VAR_TEMP
  CIP : BOOL ;	//CIP active
  UNIM : BOOL ;	//Unit Not In Maintenance
  GenRel : BOOL ;	//general OK (emergency and maintenance OK)
  EStopOK : BOOL ;	//emergency OK
  UnitNo : INT ;	//unit number
  xTmp : BOOL ;	//Temporary Bool
  iTmp : INT ;	//Temporary INT
  rTmp : REAL ;	//Temporary REAL
  dTmp : DINT ;	//Temporary DINT (free for general use)
  RetValInt : INT ;	//return value
END_VAR
BEGIN
NETWORK
TITLE =General

      SET   ;
// Simulation ---------------------------------------------------------------
      A     DB1511.DBX 1357.7;
      CC    FB  1519; // "U051Sim"
      A     DB1511.DBX   17.3;
      =     DB1511.DBX 1357.7; //Help bit for simulation

// get unit number ----------------------------------------------------------
      L     DB1510.DBW    0;
      T     #UnitNo;

// communication ------------------------------------------------------------
      UC    FB  1515; // U051Com

NETWORK
TITLE =Sequence organisation

      CLR   ;
      =     M    122.2;

// CIP Counter
      CALL FC    29 (
           UnitNo                   := #UnitNo,
           Value                    := DB1515.DBD   54,
           Enable                   := TRUE,
           Down                     := FALSE,
           OriginDetect             := 0.000000e+000,
           MaxDiffPS                := 1.000000e+000,
           SFMRec                   := DB1511.Seq.SFM[15],
           ValueOld                 := DB1511.DBD 1418);

// sequencer ----------------------------------------------------------------
      A     DB1513.DBX   43.1;
      S     DB1513.DBX   97.3;

      CALL FC    40 (
           UnitNo                   := #UnitNo);

END_FUNCTION_BLOCK

FUNCTION_BLOCK FB 1520
TITLE =U052: Water Transfer Plant 12
FAMILY : BOTEC_F1
NAME : UniA
VERSION : 2.1


VAR_TEMP
  EStopOK : BOOL ;	//auxiliary flag
  CIP : BOOL ;	//CIP Program Selected
  xTmp : BOOL ;	//Temporary Bool(free for general use)
  UnitNo : INT ;	//unit number
  UnitFB : INT ;	//unit expansion FB number
  rTmp : REAL ;	//Temporary REAL (free for general use)
  iTmp : INT ;	//Temporary INT (free for general use)
  dTmp : DINT ;	//Temporary DINT (free for general use)
END_VAR
BEGIN
NETWORK
TITLE =general

      CLR   ;
      =     #xTmp;
      =     #EStopOK;

      L     DB1520.DBW    0;
      T     #UnitNo;
      L     DB1520.DBW    2;
      T     #UnitFB;

NETWORK
TITLE =Universal value

      NOP   0;
// unv001 UnV 001 Process Status
      CALL FC    27 (
           UnitNo                   := #UnitNo,
           UnVRec                   := DB2525.unv001,
           ValExt                   := DB2525.DBD  234);

// unv002 UnV 002 Universal Value 02
      CALL FC    27 (
           UnitNo                   := #UnitNo,
           UnVRec                   := DB2525.unv002,
           ValExt                   := DB2525.DBD  362);

// unv003 UnV 003 Universal Value 03
      CALL FC    27 (
           UnitNo                   := #UnitNo,
           UnVRec                   := DB2525.unv003,
           ValExt                   := DB2525.DBD  490);

// unv004 UnV 004 Universal Value 04
      CALL FC    27 (
           UnitNo                   := #UnitNo,
           UnVRec                   := DB2525.unv004,
           ValExt                   := DB2525.DBD  618);

NETWORK
TITLE =special inputs

      NOP   0;
// U52_SpI001 SpI 001 spare
      CALL FC    14 (
           UnitNo                   := #UnitNo,
           SpIRec                   := DB2521.U52_SpI001,
           SpIBit                   := #xTmp);

NETWORK
TITLE =messages

      NOP   0;
// msg001 Msg 001 Message 01
      CALL FC    16 (
           UnitNo                   := #UnitNo,
           MsgRec                   := DB2527.msg001,
           MsgBit                   := DB2527.DBX   82.7);

// msg002 Msg 002 Message 02
      CALL FC    16 (
           UnitNo                   := #UnitNo,
           MsgRec                   := DB2527.msg002,
           MsgBit                   := DB2527.DBX  142.7);

// msg003 Msg 003 Message 03
      CALL FC    16 (
           UnitNo                   := #UnitNo,
           MsgRec                   := DB2527.msg003,
           MsgBit                   := DB2527.DBX  202.7);

NETWORK
TITLE =unit supply

      UC    FB [#UnitFB];

NETWORK
TITLE =Act1  Wasserpumpe
// Act 001
// Box           :
// Input address : #xTmp
// Output address: #xTmp
      CALL FC    70 (
           UnitNo                   := #UnitNo,
           ActRec                   := DB2520.Act1,
           Typ                      := 0,
           FBa                      := I    271.1,
           FBa2                     := #xTmp,
           Out                      := Q    271.1);

NETWORK
TITLE =A12_V11  A12 V11
// Act 002
// Box           : VSA12
// Input address : I260.6
// Output address: Q260.6
      CALL FC    70 (
           UnitNo                   := #UnitNo,
           ActRec                   := DB2520.A12_V11,
           Typ                      := 1,
           FBa                      := #xTmp,
           FBa2                     := I    260.6,
           Out                      := Q    260.6);

NETWORK
TITLE =A12_V12  A12 V12
// Act 003
// Box           : VSA12
// Input address : I260.7
// Output address: Q260.7
      CALL FC    70 (
           UnitNo                   := #UnitNo,
           ActRec                   := DB2520.A12_V12,
           Typ                      := 1,
           FBa                      := #xTmp,
           FBa2                     := I    260.7,
           Out                      := Q    260.7);

NETWORK
TITLE =A12_V13  A12 V13
// Act 004
// Box           : VSA12
// Input address : I261.0
// Output address: Q261.0
      CALL FC    70 (
           UnitNo                   := #UnitNo,
           ActRec                   := DB2520.A12_V13,
           Typ                      := 1,
           FBa                      := #xTmp,
           FBa2                     := I    261.0,
           Out                      := Q    261.0);

NETWORK
TITLE =RV1_A12
// Act 005
// Box           : Ventilinsel 2
// Input address : I321.5
// Output address: Q321.5
      CALL FC    70 (
           UnitNo                   := #UnitNo,
           ActRec                   := DB2520.RV1_A12,
           Typ                      := 1,
           FBa                      := #xTmp,
           FBa2                     := I    321.5,
           Out                      := Q    321.5);

NETWORK
TITLE =RV2_A12
// Act 006
// Box           : Ventilinsel 2
// Input address : I321.6
// Output address: Q321.6
      CALL FC    70 (
           UnitNo                   := #UnitNo,
           ActRec                   := DB2520.RV2_A12,
           Typ                      := 1,
           FBa                      := #xTmp,
           FBa2                     := I    321.6,
           Out                      := Q    321.6);

NETWORK
TITLE =RV3_A12
// Act 007
// Box           : Ventilinsel 2
// Input address : I321.7
// Output address: Q321.7
      CALL FC    70 (
           UnitNo                   := #UnitNo,
           ActRec                   := DB2520.RV3_A12,
           Typ                      := 1,
           FBa                      := #xTmp,
           FBa2                     := I    321.7,
           Out                      := Q    321.7);

NETWORK
TITLE =VR_V4
// Act 008
// Box           : Ventilinsel 4
// Input address : I336.6
// Output address: Q336.6
      CALL FC    70 (
           UnitNo                   := #UnitNo,
           ActRec                   := DB2520.VR_V4,
           Typ                      := 1,
           FBa                      := #xTmp,
           FBa2                     := I    336.6,
           Out                      := Q    336.6);

NETWORK
TITLE =U52_Act010  spare
// Act 010
// Box           :
// Output address: #xtmp
      CALL FC    70 (
           UnitNo                   := #UnitNo,
           ActRec                   := DB2520.U52_Act010,
           Typ                      := 0,
           FBa                      := #xTmp,
           FBa2                     := #xTmp,
           Out                      := #xTmp);

END_FUNCTION_BLOCK

FUNCTION_BLOCK FB 1521
TITLE =U052: Water Transfer Plant 12
FAMILY : BOTEC_F1
NAME : UniE
VERSION : 1.2


VAR_TEMP
  CIP : BOOL ;	//CIP active
  UNIM : BOOL ;	//Unit Not In Maintenance
  GenRel : BOOL ;	//general OK (emergency and maintenance OK)
  EStopOK : BOOL ;	//emergency OK
  UnitNo : INT ;	//unit number
  xTmp : BOOL ;	//Temporary Bool
  iTmp : INT ;	//Temporary INT
  rTmp : REAL ;	//Temporary REAL
  dTmp : DINT ;	//Temporary DINT (free for general use)
  RetValInt : INT ;	//return value
END_VAR
BEGIN
NETWORK
TITLE =General

      SET   ;
// Simulation ---------------------------------------------------------------
      A     DB1521.DBX 1357.7;
      CC    FB  1529; // "U052Sim"
      A     DB1521.DBX   17.3;
      =     DB1521.DBX 1357.7; //Help bit for simulation

// get unit number ----------------------------------------------------------
      L     DB1520.DBW    0;
      T     #UnitNo;

// communication ------------------------------------------------------------
      UC    FB  1525;

NETWORK
TITLE =Sequence organisation

      CLR   ;
      =     M    122.2;

// CIP Counter
      CALL FC    29 (
           UnitNo                   := #UnitNo,
           Value                    := DB1525.DBD   54,
           Enable                   := TRUE,
           Down                     := FALSE,
           OriginDetect             := 0.000000e+000,
           MaxDiffPS                := 1.000000e+000,
           SFMRec                   := DB1521.Seq.SFM[15],
           ValueOld                 := DB1521.DBD 1418);

// sequencer ----------------------------------------------------------------
      A     DB1523.DBX   43.1;
      S     DB1523.DBX   97.3;

      CALL FC    40 (
           UnitNo                   := #UnitNo);

END_FUNCTION_BLOCK

FUNCTION_BLOCK FB 1540
TITLE =U054: Water Transfer Plant 14
FAMILY : BOTEC_F1
NAME : UniA
VERSION : 2.1


VAR_TEMP
  EStopOK : BOOL ;	//auxiliary flag
  CIP : BOOL ;	//CIP Program Selected
  xTmp : BOOL ;	//Temporary Bool(free for general use)
  UnitNo : INT ;	//unit number
  UnitFB : INT ;	//unit expansion FB number
  rTmp : REAL ;	//Temporary REAL (free for general use)
  iTmp : INT ;	//Temporary INT (free for general use)
  dTmp : DINT ;	//Temporary DINT (free for general use)
END_VAR
BEGIN
NETWORK
TITLE =general

      CLR   ;
      =     #xTmp;
      =     #EStopOK;

      L     DB1540.DBW    0;
      T     #UnitNo;
      L     DB1540.DBW    2;
      T     #UnitFB;

NETWORK
TITLE =Universal value

      NOP   0;
// unv001 UnV 001 Process Status
      CALL FC    27 (
           UnitNo                   := #UnitNo,
           UnVRec                   := DB2545.unv001,
           ValExt                   := DB2545.DBD  234);

// unv002 UnV 002 Universal Value 02
      CALL FC    27 (
           UnitNo                   := #UnitNo,
           UnVRec                   := DB2545.unv002,
           ValExt                   := DB2545.DBD  362);

// unv003 UnV 003 Universal Value 03
      CALL FC    27 (
           UnitNo                   := #UnitNo,
           UnVRec                   := DB2545.unv003,
           ValExt                   := DB2545.DBD  490);

// unv004 UnV 004 Universal Value 04
      CALL FC    27 (
           UnitNo                   := #UnitNo,
           UnVRec                   := DB2545.unv004,
           ValExt                   := DB2545.DBD  618);

NETWORK
TITLE =special inputs

      NOP   0;
// U54_SpI001 SpI 001 spare
      CALL FC    14 (
           UnitNo                   := #UnitNo,
           SpIRec                   := DB2541.U54_SpI001,
           SpIBit                   := #xTmp);

NETWORK
TITLE =messages

      NOP   0;
// msg001 Msg 001 Message 01
      CALL FC    16 (
           UnitNo                   := #UnitNo,
           MsgRec                   := DB2547.msg001,
           MsgBit                   := DB2547.DBX   82.7);

// msg002 Msg 002 Message 02
      CALL FC    16 (
           UnitNo                   := #UnitNo,
           MsgRec                   := DB2547.msg002,
           MsgBit                   := DB2547.DBX  142.7);

// msg003 Msg 003 Message 03
      CALL FC    16 (
           UnitNo                   := #UnitNo,
           MsgRec                   := DB2547.msg003,
           MsgBit                   := DB2547.DBX  202.7);

NETWORK
TITLE =unit supply

      UC    FB [#UnitFB];

NETWORK
TITLE =Act1  Wasserpumpe
// Act 001
// Box           :
// Input address : #xTmp
// Output address: #xTmp
      CALL FC    70 (
           UnitNo                   := #UnitNo,
           ActRec                   := DB2540.Act1,
           Typ                      := 0,
           FBa                      := I      6.0,
           FBa2                     := #xTmp,
           Out                      := Q      6.0);

NETWORK
TITLE =A14_V11
// Act 002
// Box           : VSA14
// Input address : I96.6
// Output address: Q96.6
      CALL FC    70 (
           UnitNo                   := #UnitNo,
           ActRec                   := DB2540.A14_V11,
           Typ                      := 1,
           FBa                      := #xTmp,
           FBa2                     := I     96.6,
           Out                      := Q     96.6);

NETWORK
TITLE =A14_V12
// Act 003
// Box           : VSA14
// Input address : I96.7
// Output address: Q96.7
      CALL FC    70 (
           UnitNo                   := #UnitNo,
           ActRec                   := DB2540.A14_V12,
           Typ                      := 1,
           FBa                      := #xTmp,
           FBa2                     := I     96.7,
           Out                      := Q     96.7);

NETWORK
TITLE =A14_V13
// Act 004
// Box           : VSA14
// Input address : I97.0
// Output address: Q97.0
      CALL FC    70 (
           UnitNo                   := #UnitNo,
           ActRec                   := DB2540.A14_V13,
           Typ                      := 1,
           FBa                      := #xTmp,
           FBa2                     := I     97.0,
           Out                      := Q     97.0);

NETWORK
TITLE =RV1_A14
// Act 005
// Box           : Ventilinsel 4
// Input address : I331.5
// Output address: Q331.5
      CALL FC    70 (
           UnitNo                   := #UnitNo,
           ActRec                   := DB2540.RV1_A14,
           Typ                      := 1,
           FBa                      := #xTmp,
           FBa2                     := I    331.5,
           Out                      := Q    331.5);

NETWORK
TITLE =RV2_A14
// Act 006
// Box           : Ventilinsel 4
// Input address : I331.6
// Output address: Q331.6
      CALL FC    70 (
           UnitNo                   := #UnitNo,
           ActRec                   := DB2540.RV2_A14,
           Typ                      := 1,
           FBa                      := #xTmp,
           FBa2                     := I    331.6,
           Out                      := Q    331.6);

NETWORK
TITLE =RV3_A14
// Act 007
// Box           : Ventilinsel 4
// Input address : I331.7
// Output address: Q331.7
      CALL FC    70 (
           UnitNo                   := #UnitNo,
           ActRec                   := DB2540.RV3_A14,
           Typ                      := 1,
           FBa                      := #xTmp,
           FBa2                     := I    331.7,
           Out                      := Q    331.7);

NETWORK
TITLE =VR_V9
// Act 008
// Box           : Ventilinsel 4
// Input address : I336.1
// Output address: Q336.1
      CALL FC    70 (
           UnitNo                   := #UnitNo,
           ActRec                   := DB2540.VR_V9,
           Typ                      := 1,
           FBa                      := #xTmp,
           FBa2                     := I    336.1,
           Out                      := Q    336.1);

NETWORK
TITLE =VR_V8
// Act 009
// Box           : Ventilinsel 4
// Input address : I336.0
// Output address: Q336.0
      CALL FC    70 (
           UnitNo                   := #UnitNo,
           ActRec                   := DB2540.VR_V8,
           Typ                      := 0,//1
           FBa                      := #xTmp,
           FBa2                     := I    336.0,
           Out                      := Q    336.0);

NETWORK
TITLE =A14_V14
// Act 010
// Box           : VSA14
// Input address : I97.1
// Output address: Q97.1
      CALL FC    70 (
           UnitNo                   := #UnitNo,
           ActRec                   := DB2540.A14_V14,
           Typ                      := 0,//1
           FBa                      := #xTmp,
           FBa2                     := I     97.1,
           Out                      := Q     97.1);

END_FUNCTION_BLOCK

FUNCTION_BLOCK FB 1541
TITLE =U054: Water Transfer Plant 14
FAMILY : BOTEC_F1
NAME : UniE
VERSION : 1.2


VAR_TEMP
  CIP : BOOL ;	//CIP active
  UNIM : BOOL ;	//Unit Not In Maintenance
  GenRel : BOOL ;	//general OK (emergency and maintenance OK)
  EStopOK : BOOL ;	//emergency OK
  UnitNo : INT ;	//unit number
  xTmp : BOOL ;	//Temporary Bool
  iTmp : INT ;	//Temporary INT
  rTmp : REAL ;	//Temporary REAL
  dTmp : DINT ;	//Temporary DINT (free for general use)
  RetValInt : INT ;	//return value
END_VAR
BEGIN
NETWORK
TITLE =General

      SET   ;
// Simulation ---------------------------------------------------------------
      A     DB1541.DBX 1357.7;
      CC    FB  1549; // "U054Sim"
      A     DB1541.DBX   17.3;
      =     DB1541.DBX 1357.7; //Help bit for simulation

// get unit number ----------------------------------------------------------
      L     DB1540.DBW    0;
      T     #UnitNo;

// communication ------------------------------------------------------------
      UC    FB  1545; // U054Com

NETWORK
TITLE =Sequence organisation

      CLR   ;
      =     M    122.2;

// CIP Counter
      CALL FC    29 (
           UnitNo                   := #UnitNo,
           Value                    := DB1545.DBD   54,
           Enable                   := TRUE,
           Down                     := FALSE,
           OriginDetect             := 0.000000e+000,
           MaxDiffPS                := 1.000000e+000,
           SFMRec                   := DB1541.Seq.SFM[15],
           ValueOld                 := DB1541.DBD 1418);

// sequencer ----------------------------------------------------------------
      A     DB1543.DBX   43.1;
      S     DB1543.DBX   97.3;

      CALL FC    40 (
           UnitNo                   := #UnitNo);

NETWORK
TITLE =Werte an Mixer



END_FUNCTION_BLOCK

FUNCTION_BLOCK FB 1550
TITLE =U055: Water Transfer Plant 15
FAMILY : BOTEC_F1
NAME : UniA
VERSION : 2.1


VAR_TEMP
  EStopOK : BOOL ;	//auxiliary flag
  CIP : BOOL ;	//CIP Program Selected
  xTmp : BOOL ;	//Temporary Bool(free for general use)
  UnitNo : INT ;	//unit number
  UnitFB : INT ;	//unit expansion FB number
  rTmp : REAL ;	//Temporary REAL (free for general use)
  iTmp : INT ;	//Temporary INT (free for general use)
  dTmp : DINT ;	//Temporary DINT (free for general use)
END_VAR
BEGIN
NETWORK
TITLE =general

      CLR   ;
      =     #xTmp;
      =     #EStopOK;

      L     DB1550.DBW    0;
      T     #UnitNo;
      L     DB1550.DBW    2;
      T     #UnitFB;

NETWORK
TITLE =Universal value

      NOP   0;
// unv001 UnV 001 Process Status
      CALL FC    27 (
           UnitNo                   := #UnitNo,
           UnVRec                   := DB2555.unv001,
           ValExt                   := DB2555.DBD  234);

// unv002 UnV 002 Universal Value 02
      CALL FC    27 (
           UnitNo                   := #UnitNo,
           UnVRec                   := DB2555.unv002,
           ValExt                   := DB2555.DBD  362);

// unv003 UnV 003 Universal Value 03
      CALL FC    27 (
           UnitNo                   := #UnitNo,
           UnVRec                   := DB2555.unv003,
           ValExt                   := DB2555.DBD  490);

// unv004 UnV 004 Universal Value 04
      CALL FC    27 (
           UnitNo                   := #UnitNo,
           UnVRec                   := DB2555.unv004,
           ValExt                   := DB2555.DBD  618);

NETWORK
TITLE =special inputs

      NOP   0;
// U55_SpI001 SpI 001 spare
      CALL FC    14 (
           UnitNo                   := #UnitNo,
           SpIRec                   := DB2551.U55_SpI001,
           SpIBit                   := #xTmp);

NETWORK
TITLE =messages

      NOP   0;
// msg001 Msg 001 Message 01
      CALL FC    16 (
           UnitNo                   := #UnitNo,
           MsgRec                   := DB2557.msg001,
           MsgBit                   := DB2557.DBX   82.7);

// msg002 Msg 002 Message 02
      CALL FC    16 (
           UnitNo                   := #UnitNo,
           MsgRec                   := DB2557.msg002,
           MsgBit                   := DB2557.DBX  142.7);

// msg003 Msg 003 Message 03
      CALL FC    16 (
           UnitNo                   := #UnitNo,
           MsgRec                   := DB2557.msg003,
           MsgBit                   := DB2557.DBX  202.7);

NETWORK
TITLE =unit supply

      UC    FB [#UnitFB];

NETWORK
TITLE =Act1  Wasserpumpe
// Act 001
// Box           :
// Input address : #xTmp
// Output address: #xTmp
      CALL FC    70 (
           UnitNo                   := #UnitNo,
           ActRec                   := DB2550.Act1,
           Typ                      := 3,
           FBa                      := #xTmp,
           FBa2                     := #xTmp,
           Out                      := #xTmp);

NETWORK
TITLE =RV1_A15
// Act 005
// Box           : Ventilinsel 4
// Input address : I333.5
// Output address: Q333.5
      CALL FC    70 (
           UnitNo                   := #UnitNo,
           ActRec                   := DB2550.RV1_A15,
           Typ                      := 1,
           FBa                      := #xTmp,
           FBa2                     := I    333.5,
           Out                      := Q    333.5);

NETWORK
TITLE =RV2_A15
// Act 006
// Box           : Ventilinsel 4
// Input address : I333.6
// Output address: Q333.6
      CALL FC    70 (
           UnitNo                   := #UnitNo,
           ActRec                   := DB2550.RV2_A15,
           Typ                      := 1,
           FBa                      := #xTmp,
           FBa2                     := I    333.6,
           Out                      := Q    333.6);

NETWORK
TITLE =RV3_A15
// Act 007
// Box           : Ventilinsel 4
// Input address : I333.7
// Output address: Q333.7
      CALL FC    70 (
           UnitNo                   := #UnitNo,
           ActRec                   := DB2550.RV3_A15,
           Typ                      := 1,
           FBa                      := #xTmp,
           FBa2                     := I    333.7,
           Out                      := Q    333.7);

NETWORK
TITLE =U55_Act010  spare
// Act 010
// Box           :
// Output address: #xtmp
      CALL FC    70 (
           UnitNo                   := #UnitNo,
           ActRec                   := DB2550.U55_Act010,
           Typ                      := 0,
           FBa                      := #xTmp,
           FBa2                     := #xTmp,
           Out                      := #xTmp);

END_FUNCTION_BLOCK

FUNCTION_BLOCK FB 1551
TITLE =U055: Water Transfer Plant 15
FAMILY : BOTEC_F1
NAME : UniE
VERSION : 1.2


VAR_TEMP
  CIP : BOOL ;	//CIP active
  UNIM : BOOL ;	//Unit Not In Maintenance
  GenRel : BOOL ;	//general OK (emergency and maintenance OK)
  EStopOK : BOOL ;	//emergency OK
  UnitNo : INT ;	//unit number
  xTmp : BOOL ;	//Temporary Bool
  iTmp : INT ;	//Temporary INT
  rTmp : REAL ;	//Temporary REAL
  dTmp : DINT ;	//Temporary DINT (free for general use)
  RetValInt : INT ;	//return value
END_VAR
BEGIN
NETWORK
TITLE =General

      SET   ;
// Simulation ---------------------------------------------------------------
      A     DB1551.DBX 1357.7;
      CC    FB  1559; // "U055Sim"
      A     DB1551.DBX   17.3;
      =     DB1551.DBX 1357.7; //Help bit for simulation

// get unit number ----------------------------------------------------------
      L     DB1550.DBW    0;
      T     #UnitNo;

// communication ------------------------------------------------------------
      UC    FB  1555; // U055Com

NETWORK
TITLE =Sequence organisation

      CLR   ;
      =     M    122.2;

// CIP Counter
      CALL FC    29 (
           UnitNo                   := #UnitNo,
           Value                    := DB1555.DBD   54,
           Enable                   := TRUE,
           Down                     := FALSE,
           OriginDetect             := 0.000000e+000,
           MaxDiffPS                := 1.000000e+000,
           SFMRec                   := DB1551.Seq.SFM[15],
           ValueOld                 := DB1551.DBD 1418);

// sequencer ----------------------------------------------------------------
      A     DB1553.DBX   43.1;
      S     DB1553.DBX   97.3;

      CALL FC    40 (
           UnitNo                   := #UnitNo);

END_FUNCTION_BLOCK

FUNCTION_BLOCK FB 1560
TITLE =U056: Fresh Water Transfer
FAMILY : BOTEC_F1
NAME : UniA
VERSION : 2.1


VAR_TEMP
  EStopOK : BOOL ;	//auxiliary flag
  CIP : BOOL ;	//CIP Program Selected
  xTmp : BOOL ;	//Temporary Bool(free for general use)
  UnitNo : INT ;	//unit number
  UnitFB : INT ;	//unit expansion FB number
  rTmp : REAL ;	//Temporary REAL (free for general use)
  iTmp : INT ;	//Temporary INT (free for general use)
  dTmp : DINT ;	//Temporary DINT (free for general use)
END_VAR
BEGIN
NETWORK
TITLE =general

      CLR   ;
      =     #xTmp;
      =     #EStopOK;

      L     DB1560.DBW    0;
      T     #UnitNo;
      L     DB1560.DBW    2;
      T     #UnitFB;

NETWORK
TITLE =Universal value

      NOP   0;
// unv001 UnV 001 Process Status
      CALL FC    27 (
           UnitNo                   := #UnitNo,
           UnVRec                   := DB2565.unv001,
           ValExt                   := DB2565.DBD  234);

// unv002 UnV 002 Universal Value 02
      CALL FC    27 (
           UnitNo                   := #UnitNo,
           UnVRec                   := DB2565.unv002,
           ValExt                   := DB2565.DBD  362);

// unv003 UnV 003 Universal Value 03
      CALL FC    27 (
           UnitNo                   := #UnitNo,
           UnVRec                   := DB2565.unv003,
           ValExt                   := DB2565.DBD  490);

// unv004 UnV 004 Universal Value 04
      CALL FC    27 (
           UnitNo                   := #UnitNo,
           UnVRec                   := DB2565.unv004,
           ValExt                   := DB2565.DBD  618);

NETWORK
TITLE =messages

      NOP   0;
// msg001 Msg 001 Message 01
      CALL FC    16 (
           UnitNo                   := #UnitNo,
           MsgRec                   := DB2567.msg001,
           MsgBit                   := DB2567.DBX   82.7);

// msg002 Msg 002 Message 02
      CALL FC    16 (
           UnitNo                   := #UnitNo,
           MsgRec                   := DB2567.msg002,
           MsgBit                   := DB2567.DBX  142.7);

// msg003 Msg 003 Message 03
      CALL FC    16 (
           UnitNo                   := #UnitNo,
           MsgRec                   := DB2567.msg003,
           MsgBit                   := DB2567.DBX  202.7);

NETWORK
TITLE =unit supply

      UC    FB [#UnitFB];

NETWORK
TITLE =FW_P1  FWP1 Pumpe Frischwasser
// Act 001
// Box           : S6 U6.3
// Input address : I6.7
// Output address: Q6.7
      CALL FC    70 (
           UnitNo                   := #UnitNo,
           ActRec                   := DB2560.FW_P1,
           Typ                      := 1,
           FBa                      := #xTmp,
           FBa2                     := I      6.7,
           Out                      := Q      6.7);

NETWORK
TITLE =FW_RV2
// Act 006
// Box           : Ventilinsel 5
// Input address : I339.5
// Output address: Q339.5
      CALL FC    70 (
           UnitNo                   := #UnitNo,
           ActRec                   := DB2560.FW_RV2,
           Typ                      := 1,
           FBa                      := #xTmp,
           FBa2                     := I    339.5,
           Out                      := Q    339.5);

END_FUNCTION_BLOCK

FUNCTION_BLOCK FB 1561
TITLE =U056: Fresh Water Transfer
FAMILY : BOTEC_F1
NAME : UniE
VERSION : 1.2


VAR_TEMP
  CIP : BOOL ;	//CIP active
  UNIM : BOOL ;	//Unit Not In Maintenance
  GenRel : BOOL ;	//general OK (emergency and maintenance OK)
  EStopOK : BOOL ;	//emergency OK
  UnitNo : INT ;	//unit number
  xTmp : BOOL ;	//Temporary Bool
  iTmp : INT ;	//Temporary INT
  rTmp : REAL ;	//Temporary REAL
  dTmp : DINT ;	//Temporary DINT (free for general use)
  RetValInt : INT ;	//return value
END_VAR
BEGIN
NETWORK
TITLE =General

      SET   ;
// Simulation ---------------------------------------------------------------
      A     DB1561.DBX 1357.7;
      CC    FB  1569; // "U056Sim"
      A     DB1561.DBX   17.3;
      =     DB1561.DBX 1357.7; //Help bit for simulation

// get unit number ----------------------------------------------------------
      L     DB1560.DBW    0;
      T     #UnitNo;

// CIP ----------------------------------------------------------------------
      L     DB1561.DBD   54;
      L     0;
      <D    ;
      =     #CIP;

// emergency OK -------------------------------------------------------------
      A     DB1565.DBX   27.0; //Emergency Stop OK
      =     #EStopOK;

// Write Unit in Maintenance ------------------------------------------------

      AN    DB1561.DBX   69.7;
      =     #UNIM;

// emergency and maintenance OK ---------------------------------------------
      A     #EStopOK;
      A     #UNIM;
      =     #GenRel;

// communication ------------------------------------------------------------
      UC    FB  1565; // U056Com

NETWORK
TITLE =Universal Value

      NOP   0;

// ----------------------------------------------------------
// unv001 Process Status
// ----------------------------------------------------------
// process value to UnV
//      L     0.000000e+000
//      T     "U056UnVD".unv001.ValExt

// ----------------------------------------------------------
// unv002 Universal Value 02
// ----------------------------------------------------------
// process value to UnV
//      L     0.000000e+000
//      T     "U056UnVD".unv002.ValExt

// ----------------------------------------------------------
// unv003 Universal Value 03
// ----------------------------------------------------------
// process value to UnV
//      L     0.000000e+000
//      T     "U056UnVD".unv003.ValExt

// ----------------------------------------------------------
// unv004 Universal Value 04
// ----------------------------------------------------------
// process value to UnV
//      L     0.000000e+000
//      T     "U056UnVD".unv004.ValExt

NETWORK
TITLE =Messages

      NOP   0;

// ----------------------------------------------------------
// msg001 Message 01
// ----------------------------------------------------------
      SET   ;
      R     DB2567.DBX   80.7;
      =     DB2567.DBX   81.4;

      CLR   ;
      =     DB2567.DBX   82.7;

// ----------------------------------------------------------
// msg002 Message 02
// ----------------------------------------------------------
      SET   ;
      R     DB2567.DBX  140.7;
      =     DB2567.DBX  141.4;

      CLR   ;
      =     DB2567.DBX  142.7;

// ----------------------------------------------------------
// msg003 Message 03
// ----------------------------------------------------------
      SET   ;
      R     DB2567.DBX  200.7;
      =     DB2567.DBX  201.4;

      CLR   ;
      =     DB2567.DBX  202.7;

NETWORK
TITLE =Sequence organisation

      CLR   ;
      =     M    122.2;

// SFM supply ----------------------------------------------------------------

// sequencer ----------------------------------------------------------------
      A     DB1563.DBX   43.1;
      S     DB1563.DBX   97.3;

      CALL FC    40 (
           UnitNo                   := #UnitNo);

NETWORK
TITLE =Auto / Manual

      SET   ;
      AN    M    122.2;
      JC    MODE;
      AN    M    120.1;

// assign actuator mode
      AN    M    120.1;
      =     DB2560.DBX  105.4;
      =     DB2560.DBX  505.4;


MODE: SET   ;

NETWORK
TITLE =FW_P1 FWP1 Pumpe Frischwasser

      A     #GenRel;
      A     DB2560.DBX  106.7;
      =     DB2560.DBX  107.6;
END_FUNCTION_BLOCK

FUNCTION_BLOCK FB 1570
TITLE =U057: Water Transfer Brewhouse
FAMILY : BOTEC_F1
NAME : UniA
VERSION : 2.1


VAR_TEMP
  EStopOK : BOOL ;	//auxiliary flag
  CIP : BOOL ;	//CIP Program Selected
  xTmp : BOOL ;	//Temporary Bool(free for general use)
  UnitNo : INT ;	//unit number
  UnitFB : INT ;	//unit expansion FB number
  rTmp : REAL ;	//Temporary REAL (free for general use)
  iTmp : INT ;	//Temporary INT (free for general use)
  dTmp : DINT ;	//Temporary DINT (free for general use)
END_VAR
BEGIN
NETWORK
TITLE =general

      CLR   ;
      =     #xTmp;
      =     #EStopOK;

      L     DB1570.DBW    0;
      T     #UnitNo;
      L     DB1570.DBW    2;
      T     #UnitFB;

NETWORK
TITLE =Universal value

      NOP   0;
// unv001 UnV 001 Process Status
      CALL FC    27 (
           UnitNo                   := #UnitNo,
           UnVRec                   := DB2575.unv001,
           ValExt                   := DB2575.DBD  234);

// unv002 UnV 002 Universal Value 02
      CALL FC    27 (
           UnitNo                   := #UnitNo,
           UnVRec                   := DB2575.unv002,
           ValExt                   := DB2575.DBD  362);

// unv003 UnV 003 Universal Value 03
      CALL FC    27 (
           UnitNo                   := #UnitNo,
           UnVRec                   := DB2575.unv003,
           ValExt                   := DB2575.DBD  490);

// unv004 UnV 004 Universal Value 04
      CALL FC    27 (
           UnitNo                   := #UnitNo,
           UnVRec                   := DB2575.unv004,
           ValExt                   := DB2575.DBD  618);

NETWORK
TITLE =special inputs

      NOP   0;
// AB_SH_DT_LAMPEN_PRUEFEN SpI 002 AUSSENBEDIENUNG SUDHAUS
      CALL FC    14 (
           UnitNo                   := #UnitNo,
           SpIRec                   := DB2571.AB_SH_DT_LAMPEN_PRUEFEN,
           SpIBit                   := I     14.5);

// AB_SH_LDT_WASSER_OPUMP SpI 003 AUSSENBEDIENUNG SUDHAUS
      CALL FC    14 (
           UnitNo                   := #UnitNo,
           SpIRec                   := DB2571.AB_SH_LDT_WASSER_OPUMP,
           SpIBit                   := I     14.6);

// AB_SH_LDT_WASSER_MPUMP SpI 004 AUSSEN SUDHAUS
      CALL FC    14 (
           UnitNo                   := #UnitNo,
           SpIRec                   := DB2571.AB_SH_LDT_WASSER_MPUMP,
           SpIBit                   := I     15.3);

// AB_SH_DT_START SpI 005 AUSSENBEDIENUNG SUDHAUS
      CALL FC    14 (
           UnitNo                   := #UnitNo,
           SpIRec                   := DB2571.AB_SH_DT_START,
           SpIBit                   := I     15.6);

// AB_SH_DT_STOP SpI 006 AUSSENBEDIENUNG SUDHAUS
      CALL FC    14 (
           UnitNo                   := #UnitNo,
           SpIRec                   := DB2571.AB_SH_DT_STOP,
           SpIBit                   := I     15.7);

NETWORK
TITLE =messages

      NOP   0;
// msg001 Msg 001 Message 01
      CALL FC    16 (
           UnitNo                   := #UnitNo,
           MsgRec                   := DB2577.msg001,
           MsgBit                   := DB2577.DBX   82.7);

// msg002 Msg 002 Message 02
      CALL FC    16 (
           UnitNo                   := #UnitNo,
           MsgRec                   := DB2577.msg002,
           MsgBit                   := DB2577.DBX  142.7);

// msg003 Msg 003 Message 03
      CALL FC    16 (
           UnitNo                   := #UnitNo,
           MsgRec                   := DB2577.msg003,
           MsgBit                   := DB2577.DBX  202.7);

NETWORK
TITLE =unit supply

      UC    FB [#UnitFB];

NETWORK
TITLE =SH_P1  SHP1
// Act 001
// Box           : S6 U6.3
// Input address : I6.4
// Output address: Q6.4
      CALL FC    70 (
           UnitNo                   := #UnitNo,
           ActRec                   := DB2570.SH_P1,
           Typ                      := 1,
           FBa                      := #xTmp,
           FBa2                     := I      6.4,
           Out                      := Q      6.4);

NETWORK
TITLE =AB_SH_LAMPE_LDT_WASSOP  Lampe AUSSEN SUDHAUS (ohne Pumpe)
// Act 002
// Box           : S6 U6.3
// Output address: Q14.6
      CALL FC    70 (
           UnitNo                   := #UnitNo,
           ActRec                   := DB2570.AB_SH_LAMPE_LDT_WASSOP,
           Typ                      := 0,
           FBa                      := #xTmp,
           FBa2                     := #xTmp,
           Out                      := Q     14.6);

NETWORK
TITLE =AB_SH_LAMPE_FREIGWASSER  Lampe AUSSENBEDIENUNG SUDHAUS (Freigabe
// Act 003
// Box           : S6 U6.3
// Output address: Q14.7
      CALL FC    70 (
           UnitNo                   := #UnitNo,
           ActRec                   := DB2570.AB_SH_LAMPE_FREIGWASSER,
           Typ                      := 0,
           FBa                      := #xTmp,
           FBa2                     := #xTmp,
           Out                      := Q     14.7);

NETWORK
TITLE =AB_SH_LAMPE_LDT_WASSMP  Lampe AUSSENBEDIENUNG SUDHAUS (mit Pumpe
// Act 004
// Box           : S6 U6.3
// Output address: Q15.0
      CALL FC    70 (
           UnitNo                   := #UnitNo,
           ActRec                   := DB2570.AB_SH_LAMPE_LDT_WASSMP,
           Typ                      := 0,
           FBa                      := #xTmp,
           FBa2                     := #xTmp,
           Out                      := Q     15.0);

NETWORK
TITLE =BH_RV2
// Act 006
// Box           : Ventilinsel 5
// Input address : I339.6
// Output address: Q339.6
      CALL FC    70 (
           UnitNo                   := #UnitNo,
           ActRec                   := DB2570.BH_RV2,
           Typ                      := 1,
           FBa                      := #xTmp,
           FBa2                     := I    339.6,
           Out                      := Q    339.6);

END_FUNCTION_BLOCK

FUNCTION_BLOCK FB 1571
TITLE =U057: Water Transfer Brewhouse
FAMILY : BOTEC_F1
NAME : UniE
VERSION : 1.2


VAR_TEMP
  CIP : BOOL ;	//CIP active
  UNIM : BOOL ;	//Unit Not In Maintenance
  GenRel : BOOL ;	//general OK (emergency and maintenance OK)
  EStopOK : BOOL ;	//emergency OK
  UnitNo : INT ;	//unit number
  xTmp : BOOL ;	//Temporary Bool
  iTmp : INT ;	//Temporary INT
  rTmp : REAL ;	//Temporary REAL
  dTmp : DINT ;	//Temporary DINT (free for general use)
  RetValInt : INT ;	//return value
END_VAR
BEGIN
NETWORK
TITLE =General

      SET   ;
// Simulation ---------------------------------------------------------------
      A     DB1571.DBX 1357.7;
      CC    FB  1579; // "U057Sim"
      A     DB1571.DBX   17.3;
      =     DB1571.DBX 1357.7; //Help bit for simulation

// get unit number ----------------------------------------------------------
      L     DB1570.DBW    0;
      T     #UnitNo;

// CIP ----------------------------------------------------------------------
      L     DB1571.DBD   54;
      L     0;
      <D    ;
      =     #CIP;

// emergency OK -------------------------------------------------------------
      A     DB1575.DBX   27.0; //Emergency Stop OK
      =     #EStopOK;

// Write Unit in Maintenance ------------------------------------------------

      AN    DB1571.DBX   69.7;
      =     #UNIM;

// emergency and maintenance OK ---------------------------------------------
      A     #EStopOK;
      A     #UNIM;
      =     #GenRel;

// communication ------------------------------------------------------------
      UC    FB  1575; // U057Com

NETWORK
TITLE =Universal Value

      NOP   0;

// ----------------------------------------------------------
// unv001 Process Status
// ----------------------------------------------------------
// process value to UnV
//      L     0.000000e+000
//      T     "U057UnVD".unv001.ValExt

// ----------------------------------------------------------
// unv002 Universal Value 02
// ----------------------------------------------------------
// process value to UnV
//      L     0.000000e+000
//      T     "U057UnVD".unv002.ValExt

// ----------------------------------------------------------
// unv003 Universal Value 03
// ----------------------------------------------------------
// process value to UnV
//      L     0.000000e+000
//      T     "U057UnVD".unv003.ValExt

// ----------------------------------------------------------
// unv004 Universal Value 04
// ----------------------------------------------------------
// process value to UnV
//      L     0.000000e+000
//      T     "U057UnVD".unv004.ValExt

NETWORK
TITLE =Special Input

      NOP   0;

// ----------------------------------------------------------
// AB_SH_DT_LAMPEN_PRUEFEN AUSSENBEDIENUNG SUDHAUS
// ----------------------------------------------------------
      CLR   ;
//      =     "U057SpID".AB_SH_DT_LAMPEN_PRUEFEN.EAl
//      =     "U057SpID".AB_SH_DT_LAMPEN_PRUEFEN.Pre

// ----------------------------------------------------------
// AB_SH_LDT_WASSER_OPUMP AUSSENBEDIENUNG SUDHAUS
// ----------------------------------------------------------
      CLR   ;
//      =     "U057SpID".AB_SH_LDT_WASSER_OPUMP.EAl
//      =     "U057SpID".AB_SH_LDT_WASSER_OPUMP.Pre

// ----------------------------------------------------------
// AB_SH_LDT_WASSER_MPUMP AUSSENBEDIENUNG SUDHAUS
// ----------------------------------------------------------
      CLR   ;
//      =     "U057SpID".AB_SH_LDT_WASSER_MPUMP.EAl
//      =     "U057SpID".AB_SH_LDT_WASSER_MPUMP.Pre

// ----------------------------------------------------------
// AB_SH_DT_START AUSSENBEDIENUNG SUDHAUS
// ----------------------------------------------------------
      CLR   ;
//      =     "U057SpID".AB_SH_DT_START.EAl
//      =     "U057SpID".AB_SH_DT_START.Pre

// ----------------------------------------------------------
// AB_SH_DT_STOP AUSSENBEDIENUNG SUDHAUS
// ----------------------------------------------------------
      CLR   ;
//      =     "U057SpID".AB_SH_DT_STOP.EAl
//      =     "U057SpID".AB_SH_DT_STOP.Pre

NETWORK
TITLE =Messages

      NOP   0;

// ----------------------------------------------------------
// msg001 Message 01
// ----------------------------------------------------------
      SET   ;
      R     DB2577.DBX   80.7;
      =     DB2577.DBX   81.4;

      CLR   ;
      =     DB2577.DBX   82.7;

// ----------------------------------------------------------
// msg002 Message 02
// ----------------------------------------------------------
      SET   ;
      R     DB2577.DBX  140.7;
      =     DB2577.DBX  141.4;

      CLR   ;
      =     DB2577.DBX  142.7;

// ----------------------------------------------------------
// msg003 Message 03
// ----------------------------------------------------------
      SET   ;
      R     DB2577.DBX  200.7;
      =     DB2577.DBX  201.4;

      CLR   ;
      =     DB2577.DBX  202.7;

NETWORK
TITLE =Sequence organisation


// SFM supply ----------------------------------------------------------------

// sequencer ----------------------------------------------------------------
      A     DB1573.DBX   43.1;
      S     DB1573.DBX   97.3;

      CALL FC    40 (
           UnitNo                   := #UnitNo);

NETWORK
TITLE =Auto / Manual

      SET   ;
      AN    M    122.2;
      JC    MODE;
      AN    M    120.1;

// assign actuator mode
      AN    M    120.1;
      =     DB2570.DBX  105.4;
      =     DB2570.DBX  185.4;
      =     DB2570.DBX  265.4;
      =     DB2570.DBX  345.4;

      =     DB2570.DBX  425.4;
      =     DB2570.DBX  505.4;




MODE: SET   ;

NETWORK
TITLE =SH_P1 SHP1
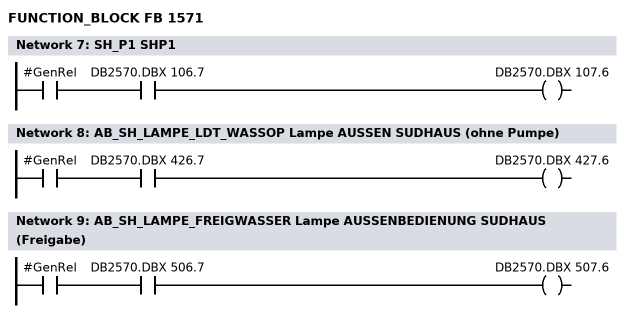

      A     #GenRel;
      A     DB2570.DBX  106.7;
      =     DB2570.DBX  107.6;
NETWORK
TITLE =AB_SH_LAMPE_LDT_WASSOP Lampe AUSSEN SUDHAUS (ohne Pumpe)

      A     #GenRel;
      A     DB2570.DBX  426.7;
      =     DB2570.DBX  427.6;
NETWORK
TITLE =AB_SH_LAMPE_FREIGWASSER Lampe AUSSENBEDIENUNG SUDHAUS (Freigabe)

      A     #GenRel;
      A     DB2570.DBX  506.7;
      =     DB2570.DBX  507.6;
END_FUNCTION_BLOCK

FUNCTION_BLOCK FB 1580
TITLE =U058: Water Transfer Syrup
FAMILY : BOTEC_F1
NAME : UniA
VERSION : 2.1


VAR_TEMP
  EStopOK : BOOL ;	//auxiliary flag
  CIP : BOOL ;	//CIP Program Selected
  xTmp : BOOL ;	//Temporary Bool(free for general use)
  UnitNo : INT ;	//unit number
  UnitFB : INT ;	//unit expansion FB number
  rTmp : REAL ;	//Temporary REAL (free for general use)
  iTmp : INT ;	//Temporary INT (free for general use)
  dTmp : DINT ;	//Temporary DINT (free for general use)
END_VAR
BEGIN
NETWORK
TITLE =general

      CLR   ;
      =     #xTmp;
      =     #EStopOK;

      L     DB1580.DBW    0;
      T     #UnitNo;
      L     DB1580.DBW    2;
      T     #UnitFB;

NETWORK
TITLE =analog inputs

      NOP   0;
// SRW_PIC1 AnI 001
      CALL FC    24 (
           UnitNo                   := #UnitNo,
           AnIRec                   := DB2583.SRW_PIC1,
           ValPer                   := IW   516);

NETWORK
TITLE =Universal value

      NOP   0;
// unv001 UnV 001 Process Status
      CALL FC    27 (
           UnitNo                   := #UnitNo,
           UnVRec                   := DB2585.unv001,
           ValExt                   := DB2585.DBD  234);

// unv002 UnV 002 Universal Value 02
      CALL FC    27 (
           UnitNo                   := #UnitNo,
           UnVRec                   := DB2585.unv002,
           ValExt                   := DB2585.DBD  362);

// unv003 UnV 003 Universal Value 03
      CALL FC    27 (
           UnitNo                   := #UnitNo,
           UnVRec                   := DB2585.unv003,
           ValExt                   := DB2585.DBD  490);

// unv004 UnV 004 Universal Value 04
      CALL FC    27 (
           UnitNo                   := #UnitNo,
           UnVRec                   := DB2585.unv004,
           ValExt                   := DB2585.DBD  618);

NETWORK
TITLE =special inputs

      NOP   0;
// SW_FS1 SpI 002 Flussschalter Wasserpumpe Sirupraum
      CALL FC    14 (
           UnitNo                   := #UnitNo,
           SpIRec                   := DB2581.SW_FS1,
           SpIBit                   := I    188.0);

// WAS_Anforderung SpI 003 Anforderung Wasser
      CALL FC    14 (
           UnitNo                   := #UnitNo,
           SpIRec                   := DB2581.WAS_Anforderung,
           SpIBit                   := DB1585.DBX   26.3);

NETWORK
TITLE =messages

      NOP   0;
// msg001 Msg 001 Message 01
      CALL FC    16 (
           UnitNo                   := #UnitNo,
           MsgRec                   := DB2587.msg001,
           MsgBit                   := DB2587.DBX   82.7);

// msg002 Msg 002 Message 02
      CALL FC    16 (
           UnitNo                   := #UnitNo,
           MsgRec                   := DB2587.msg002,
           MsgBit                   := DB2587.DBX  142.7);

// msg003 Msg 003 Message 03
      CALL FC    16 (
           UnitNo                   := #UnitNo,
           MsgRec                   := DB2587.msg003,
           MsgBit                   := DB2587.DBX  202.7);

NETWORK
TITLE =controllers

      NOP   0;
// SR_P1_PID PID 001 Druckregelung Sirupwasser SR.P1
      CALL FC    55 (
           UnitNo                   := #UnitNo,
           PIDRec                   := DB2586.SR_P1_PID,
           SpExt                    := DB2586.DBD  234,
           PVal                     := DB2586.DBD  254,
           OPer                     := PQW  516);

NETWORK
TITLE =unit supply

      UC    FB [#UnitFB];

NETWORK
TITLE =SR_P1  Wasserpumpe Sirupraum
// Act 001
// Box           : VSSK
// Input address : I73.7
// Output address: Q53.7
      CALL FC    70 (
           UnitNo                   := #UnitNo,
           ActRec                   := DB2580.SR_P1,
           Typ                      := 3,
           FBa                      := I     73.7,
           FBa2                     := #xTmp,
           Out                      := Q     53.7);

NETWORK
TITLE =WAS_Bereit  Wasser kann agefordert werden
// Act 002
// Box           : Sirup
// Output address: DB_SEND_DOEHLER.Wasser.Bereit
      CALL FC    70 (
           UnitNo                   := #UnitNo,
           ActRec                   := DB2580.WAS_Bereit,
           Typ                      := 0,
           FBa                      := #xTmp,
           FBa2                     := #xTmp,
           Out                      := DB404.DBX    2.0);

NETWORK
TITLE =WAS_Pumpe_laeuft  Die Wasserpumpe laeuft
// Act 003
// Box           : Sirup
// Output address: DB_SEND_DOEHLER.Wasser.Pumpe_laeuft
      CALL FC    70 (
           UnitNo                   := #UnitNo,
           ActRec                   := DB2580.WAS_Pumpe_laeuft,
           Typ                      := 0,
           FBa                      := #xTmp,
           FBa2                     := #xTmp,
           Out                      := DB404.DBX    2.1);

NETWORK
TITLE =SK_RV2
// Act 006
// Box           : Ventilinsel 5
// Input address : I339.4
// Output address: Q339.4
      CALL FC    70 (
           UnitNo                   := #UnitNo,
           ActRec                   := DB2580.SK_RV2,
           Typ                      := 1,
           FBa                      := #xTmp,
           FBa2                     := I    339.4,
           Out                      := Q    339.4);

END_FUNCTION_BLOCK

FUNCTION_BLOCK FB 1581
TITLE =U058: Water Transfer Syrup
FAMILY : BOTEC_F1
NAME : UniE
VERSION : 1.2


VAR_TEMP
  CIP : BOOL ;	//CIP active
  UNIM : BOOL ;	//Unit Not In Maintenance
  GenRel : BOOL ;	//general OK (emergency and maintenance OK)
  EStopOK : BOOL ;	//emergency OK
  UnitNo : INT ;	//unit number
  xTmp : BOOL ;	//Temporary Bool
  iTmp : INT ;	//Temporary INT
  rTmp : REAL ;	//Temporary REAL
  dTmp : DINT ;	//Temporary DINT (free for general use)
  RetValInt : INT ;	//return value
END_VAR
BEGIN
NETWORK
TITLE =General

      SET   ;
// Simulation ---------------------------------------------------------------
      A     DB1581.DBX 1357.7;
      CC    FB  1589; // "U058Sim"
      A     DB1581.DBX   17.3;
      =     DB1581.DBX 1357.7; //Help bit for simulation

// get unit number ----------------------------------------------------------
      L     DB1580.DBW    0;
      T     #UnitNo;

// CIP ----------------------------------------------------------------------
      L     DB1581.DBD   54;
      L     0;
      <D    ;
      =     #CIP;

// emergency OK -------------------------------------------------------------
      A     DB1585.DBX   27.0; //Emergency Stop OK
      =     #EStopOK;

// Write Unit in Maintenance ------------------------------------------------

      AN    DB1581.DBX   69.7;
      =     #UNIM;

// emergency and maintenance OK ---------------------------------------------
      A     #EStopOK;
      A     #UNIM;
      =     #GenRel;

// communication ------------------------------------------------------------
      UC    FB  1585; // U058Com

NETWORK
TITLE =Analog Inputs

      NOP   0;

// ----------------------------------------------------------
// SRW_PIC1
// ----------------------------------------------------------
      L     DB1581.DBD 1118; // !!! insert correct SFM !!!
      T     DB2583.DBD  238;

      SET   ;
      =     DB2583.DBX  141.5;

NETWORK
TITLE =Universal Value

      NOP   0;

// ----------------------------------------------------------
// unv001 Process Status
// ----------------------------------------------------------
// process value to UnV
//      L     0.000000e+000
//      T     "U058UnVD".unv001.ValExt

// ----------------------------------------------------------
// unv002 Universal Value 02
// ----------------------------------------------------------
// process value to UnV
//      L     0.000000e+000
//      T     "U058UnVD".unv002.ValExt

// ----------------------------------------------------------
// unv003 Universal Value 03
// ----------------------------------------------------------
// process value to UnV
//      L     0.000000e+000
//      T     "U058UnVD".unv003.ValExt

// ----------------------------------------------------------
// unv004 Universal Value 04
// ----------------------------------------------------------
// process value to UnV
//      L     0.000000e+000
//      T     "U058UnVD".unv004.ValExt

NETWORK
TITLE =Special Input

      NOP   0;

// ----------------------------------------------------------
// SW_FS1 Flussschalter Wasserpumpe Sirupraum
// ----------------------------------------------------------
      A     DB2580.DBX  102.6;
      =     DB2581.DBX  141.4;
      =     DB2581.DBX  141.5;

// ----------------------------------------------------------
// WAS_Anforderung Anforderung Wasser
// ----------------------------------------------------------
      CLR   ;
      =     DB2581.DBX  201.4;
      =     DB2581.DBX  201.5;

NETWORK
TITLE =Messages

      NOP   0;

// ----------------------------------------------------------
// msg001 Message 01
// ----------------------------------------------------------
      SET   ;
      R     DB2587.DBX   80.7;
      =     DB2587.DBX   81.4;

      CLR   ;
      =     DB2587.DBX   82.7;

// ----------------------------------------------------------
// msg002 Message 02
// ----------------------------------------------------------
      SET   ;
      R     DB2587.DBX  140.7;
      =     DB2587.DBX  141.4;

      CLR   ;
      =     DB2587.DBX  142.7;

// ----------------------------------------------------------
// msg003 Message 03
// ----------------------------------------------------------
      SET   ;
      R     DB2587.DBX  200.7;
      =     DB2587.DBX  201.4;

      CLR   ;
      =     DB2587.DBX  202.7;

NETWORK
TITLE =PID controller
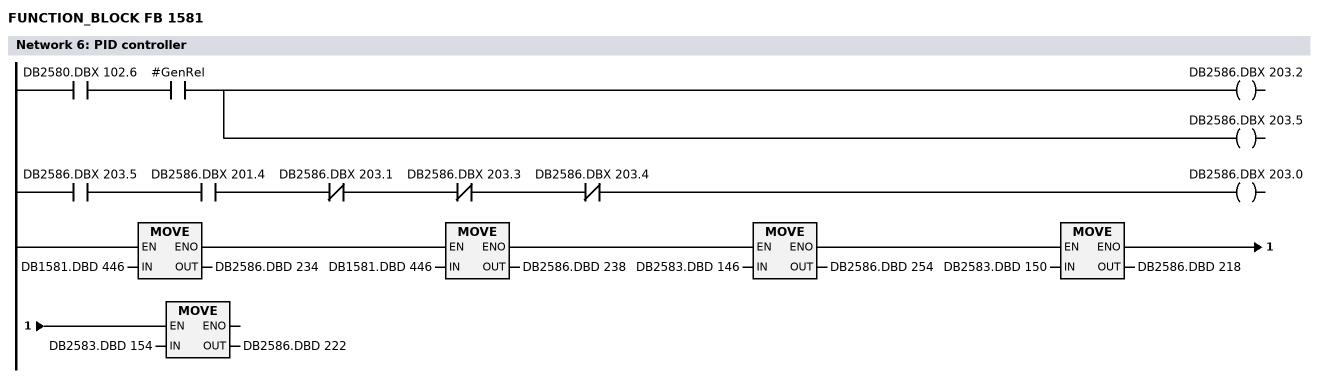

      NOP   0;

// ----------------------------------------------------------
// SR_P1_PID Druckregelung Sirupwasser SR.P1
// ----------------------------------------------------------
// starting value -----------------------
      A     DB2580.DBX  102.6;
      A     #GenRel;
      =     DB2586.DBX  203.2;
      =     DB2586.DBX  203.5;

// enable alarm -------------------------
      A     DB2586.DBX  203.5;
      A     DB2586.DBX  201.4;
      AN    DB2586.DBX  203.1;
      AN    DB2586.DBX  203.3;
      AN    DB2586.DBX  203.4;
      =     DB2586.DBX  203.0;

// setpoint to controller ---------------
      L     DB1581.DBD  446;
      T     DB2586.DBD  234;

// static value to controller ----------
      L     DB1581.DBD  446;
      T     DB2586.DBD  238;

// process value to controller ----------
      L     DB2583.DBD  146;
      T     DB2586.DBD  254;

// low/high value to controller ---------
      L     DB2583.DBD  150;
      T     DB2586.DBD  218;

      L     DB2583.DBD  154;
      T     DB2586.DBD  222;

NETWORK
TITLE =Sequence organisation

      CLR   ;
      =     M    122.2;

// SFM supply ----------------------------------------------------------------

// analog value to SFM  -----------------------
      L     DB2583.DBD  146;
      T     DB1581.DBD  450;

// sequencer ----------------------------------------------------------------
      A     DB1583.DBX   43.1;
      S     DB1583.DBX   97.3;

      CALL FC    40 (
           UnitNo                   := #UnitNo);

NETWORK
TITLE =Auto / Manual

      SET   ;
      AN    M    122.2;
      JC    MODE;
      AN    M    120.1;

// assign actuator mode
      AN    M    120.1;
      =     DB2580.DBX  105.4;
      =     DB2580.DBX  185.4;
      =     DB2580.DBX  265.4;
      =     DB2580.DBX  505.4;

// assign PID mode
      S     DB2586.DBX  201.4;
      S     DB2586.DBX  201.5;


MODE: SET   ;

NETWORK
TITLE =SR_P1 Wasserpumpe Sirupraum
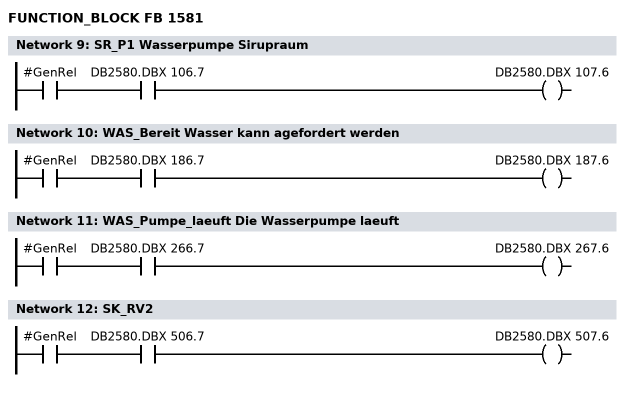

      A     #GenRel;
      A     DB2580.DBX  106.7;
      =     DB2580.DBX  107.6;
NETWORK
TITLE =WAS_Bereit Wasser kann agefordert werden

      A     #GenRel;
      A     DB2580.DBX  186.7;
      =     DB2580.DBX  187.6;
NETWORK
TITLE =WAS_Pumpe_laeuft Die Wasserpumpe laeuft

      A     #GenRel;
      A     DB2580.DBX  266.7;
      =     DB2580.DBX  267.6;
NETWORK
TITLE =SK_RV2

      A     #GenRel;
      A     DB2580.DBX  506.7;
      =     DB2580.DBX  507.6;
END_FUNCTION_BLOCK

FUNCTION_BLOCK FB 1590
TITLE =U059: Molchwasser
FAMILY : BOTEC_F1
NAME : U059A
VERSION : 2.1


VAR_TEMP
  EStopOK : BOOL ;	//auxiliary flag
  CIP : BOOL ;	//CIP Program Selected
  xTmp : BOOL ;	//Temporary Bool(free for general use)
  DummyBool : BOOL ;	//Temporary Bool(free for general use)
  UnitNo : INT ;	//unit number
  UnitFB : INT ;	//unit expansion FB number
  rTmp : REAL ;	//Temporary REAL (free for general use)
  iTmp : INT ;	//Temporary INT (free for general use)
  DummyInt : INT ;	//Temporary INT (free for general use)
  dTmp : DINT ;	//Temporary DINT (free for general use)
END_VAR
BEGIN
NETWORK
TITLE =general

      CLR   ;
      =     #xTmp;
      =     #EStopOK;

      L     DB1590.DBW    0;
      T     #UnitNo;
      L     DB1590.DBW    2;
      T     #UnitFB;

NETWORK
TITLE =Universal value

      NOP   0;
// C_UnV001 UnV 001 Prozessstatuss
      CALL FC    27 (
           UnitNo                   := #UnitNo,
           UnVRec                   := DB2595.C_UnV001,
           ValExt                   := DB2595.DBD  234);

// C_UnV002 UnV 002 spare
      CALL FC    27 (
           UnitNo                   := #UnitNo,
           UnVRec                   := DB2595.C_UnV002,
           ValExt                   := DB2595.DBD  362);

NETWORK
TITLE =special inputs

      NOP   0;
// GOA_SKP1 SpI 004 GOA
      CALL FC    14 (
           UnitNo                   := #UnitNo,
           SpIRec                   := DB2591.GOA_SKP1,
           SpIBit                   := I    264.2);

// GOA_SRGV SpI 005 GOA Molchw. Gully
      CALL FC    14 (
           UnitNo                   := #UnitNo,
           SpIRec                   := DB2591.GOA_SRGV,
           SpIBit                   := I    264.4);

NETWORK
TITLE =messages

      NOP   0;
// C_Msg002 Msg 002 spare
      CALL FC    16 (
           UnitNo                   := #UnitNo,
           MsgRec                   := DB2597.C_Msg002,
           MsgBit                   := DB2597.DBX  142.7);

NETWORK
TITLE =unit supply

      UC    FB [#UnitFB];
NETWORK
TITLE =MW_GK1  MOLCHE SR Reserve
// Act 003
// Box           : VS-SRA
// Input address : I191.0
// Output address: Q191.0
      CALL FC    70 (
           UnitNo                   := #UnitNo,
           ActRec                   := DB2590.MW_GK1,
           Typ                      := 1,
           FBa                      := #xTmp,
           FBa2                     := I    191.0,
           Out                      := Q    191.0);

NETWORK
TITLE =VR_MWV  MOLCHE SR
// Act 004
// Box           : VS-SRA
// Input address : I191.1
// Output address: Q191.1
      CALL FC    70 (
           UnitNo                   := #UnitNo,
           ActRec                   := DB2590.VR_MWV,
           Typ                      := 1,
           FBa                      := #xTmp,
           FBa2                     := I    191.1,
           Out                      := Q    191.1);

END_FUNCTION_BLOCK

FUNCTION_BLOCK FB 1591
TITLE =U059: Molchwasser
FAMILY : BOTEC_F1
NAME : U059E
VERSION : 1.2


VAR_TEMP
  CIP : BOOL ;	//CIP active
  UNIM : BOOL ;	//Unit Not In Maintenance
  GenRel : BOOL ;	//general OK (emergency and maintenance OK)
  EStopOK : BOOL ;	//emergency OK
  UnitNo : INT ;	//unit number
  xTmp : BOOL ;	//Temporary Bool
  iTmp : INT ;	//Temporary INT
  rTmp : REAL ;	//Temporary REAL
  dTmp : DINT ;	//Temporary DINT (free for general use)
  RetValInt : INT ;	//return value
END_VAR
BEGIN
NETWORK
TITLE =General

      SET   ;
// Simulation ---------------------------------------------------------------
      A     DB1591.DBX 1357.7;
      CC    FB  1599; // "U059Sim"
      A     DB1591.DBX   17.3;
      =     DB1591.DBX 1357.7; //Help bit for simulation

// get unit number ----------------------------------------------------------
      L     DB1590.DBW    0;
      T     #UnitNo;

// CIP ----------------------------------------------------------------------
      L     DB1591.DBD   54;
      L     0;
      <D    ;
      =     #CIP;

// emergency OK -------------------------------------------------------------
      A     DB1595.DBX   27.0; //Emergency Stop OK
      =     #EStopOK;

// Write Unit in Maintenance ------------------------------------------------

      AN    DB1591.DBX   69.7;
      =     #UNIM;

// emergency and maintenance OK ---------------------------------------------
      A     #EStopOK;
      A     #UNIM;
      =     #GenRel;

// communication ------------------------------------------------------------
      UC    FB  1595; // U059Com

NETWORK
TITLE =Universal Value

      NOP   0;

// ----------------------------------------------------------
// C_UnV001 Prozessstatuss
// ----------------------------------------------------------
// process value to UnV
//      L     0.000000e+000
//      T     "U059UnVD".C_UnV001.ValExt

// ----------------------------------------------------------
// C_UnV002 spare
// ----------------------------------------------------------
// process value to UnV
//      L     0.000000e+000
//      T     "U059UnVD".C_UnV002.ValExt

NETWORK
TITLE =Special Input

      NOP   0;

// ----------------------------------------------------------
// GOA_SKP1 GOA
// ----------------------------------------------------------
      SET   ;
      =     DB2591.DBX  261.4;
      =     DB2591.DBX  261.5;

// ----------------------------------------------------------
// GOA_SRGV GOA Molchw. Gully
// ----------------------------------------------------------
      SET   ;
      =     DB2591.DBX  321.4;
      =     DB2591.DBX  321.5;

NETWORK
TITLE =Messages

      NOP   0;

// ----------------------------------------------------------
// C_Msg002 spare
// ----------------------------------------------------------
      SET   ;
      R     DB2597.DBX  140.7;
      =     DB2597.DBX  141.4;

      CLR   ;
      =     DB2597.DBX  142.7;

NETWORK
TITLE =Sequence organisation

      CLR   ;
      =     M    122.2;

// SFM supply ----------------------------------------------------------------

// sequencer ----------------------------------------------------------------
      A     DB1593.DBX   43.1;
      S     DB1593.DBX   97.3;

      CALL FC    40 (
           UnitNo                   := #UnitNo);

NETWORK
TITLE =Auto / Manual

      SET   ;
      AN    M    122.2;
      JC    MODE;
      AN    M    120.1;

// assign actuator mode
      AN    M    120.1;
      =     DB2590.DBX  265.4;
      =     DB2590.DBX  345.4;



MODE: SET   ;

NETWORK
TITLE =MW_GK1 MOLCHE SR Reserve
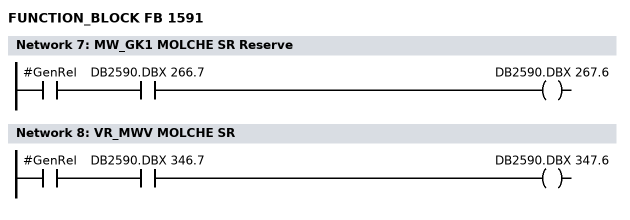

      A     #GenRel;
      A     DB2590.DBX  266.7;
      =     DB2590.DBX  267.6;
NETWORK
TITLE =VR_MWV MOLCHE SR

      A     #GenRel;
      A     DB2590.DBX  346.7;
      =     DB2590.DBX  347.6;
END_FUNCTION_BLOCK

FUNCTION_BLOCK FB 1630
TITLE =U063: Abfüllanlage  3
FAMILY : BOTEC_F1
NAME : U063A
VERSION : 2.1


VAR_TEMP
  EStopOK : BOOL ;	//auxiliary flag
  CIP : BOOL ;	//CIP Program Selected
  xTmp : BOOL ;	//Temporary Bool(free for general use)
  DummyBool : BOOL ;	//Temporary Bool(free for general use)
  UnitNo : INT ;	//unit number
  UnitFB : INT ;	//unit expansion FB number
  rTmp : REAL ;	//Temporary REAL (free for general use)
  iTmp : INT ;	//Temporary INT (free for general use)
  DummyInt : INT ;	//Temporary INT (free for general use)
  dTmp : DINT ;	//Temporary DINT (free for general use)
END_VAR
BEGIN
NETWORK
TITLE =general

      CLR   ;
      =     #xTmp;
      =     #EStopOK;

      L     DB1630.DBW    0;
      T     #UnitNo;
      L     DB1630.DBW    2;
      T     #UnitFB;

NETWORK
TITLE =analog inputs

      NOP   0;
// KEG_MIXER_KZE_NIVEAU AnI 001 KEG Mixer/KZE Niveau Steriltank
      CALL FC    24 (
           UnitNo                   := #UnitNo,
           AnIRec                   := DB2633.KEG_MIXER_KZE_NIVEAU,
           ValPer                   := PIW  954);

// KEG_MIXER_KZE_SORTE AnI 002 KEG Mixer/KZE Sortennummer Produkt
      CALL FC    24 (
           UnitNo                   := #UnitNo,
           AnIRec                   := DB2633.KEG_MIXER_KZE_SORTE,
           ValPer                   := PIW  952);

NETWORK
TITLE =Universal value

      NOP   0;
// unv001 UnV 001 Process Status
      CALL FC    27 (
           UnitNo                   := #UnitNo,
           UnVRec                   := DB2635.unv001,
           ValExt                   := DB2635.DBD  234);

// unv002 UnV 002 Universal Value 02
      CALL FC    27 (
           UnitNo                   := #UnitNo,
           UnVRec                   := DB2635.unv002,
           ValExt                   := DB2635.DBD  362);

// KEG_MIXER_PROGRAMMNR UnV 003 Preselection 1/2/3 GES./GES.without KZE/KZE
      CALL FC    27 (
           UnitNo                   := #UnitNo,
           UnVRec                   := DB2635.KEG_MIXER_PROGRAMMNR,
           ValExt                   := DB2635.DBD  490);

// KEG_MIXER_TANKNUMMER UnV 004 Tank number clean water tank [1..9]
      CALL FC    27 (
           UnitNo                   := #UnitNo,
           UnVRec                   := DB2635.KEG_MIXER_TANKNUMMER,
           ValExt                   := DB2635.DBD  618);

NETWORK
TITLE =special inputs

      NOP   0;
// KEG_MIXER_CIP_BEREIT SpI 003 KEG Mixer/KZE CIP Bereit
      CALL FC    14 (
           UnitNo                   := #UnitNo,
           SpIRec                   := DB2631.KEG_MIXER_CIP_BEREIT,
           SpIBit                   := I    946.1);

// KEG_MIXER_VOLL SpI 004 KEG Mixer/KZE Vollmeldung
      CALL FC    14 (
           UnitNo                   := #UnitNo,
           SpIRec                   := DB2631.KEG_MIXER_VOLL,
           SpIBit                   := I    946.2);

// KEG_MIXER_LEER SpI 005 KEG Mixer/KZE Leermeldung
      CALL FC    14 (
           UnitNo                   := #UnitNo,
           SpIRec                   := DB2631.KEG_MIXER_LEER,
           SpIBit                   := I    946.3);

// KEG_FUELLER_CIP_BEREIT SpI 007 KEG Füller CIP Bereitschaft
      CALL FC    14 (
           UnitNo                   := #UnitNo,
           SpIRec                   := DB2631.KEG_FUELLER_CIP_BEREIT,
           SpIBit                   := I    986.1);

// KEG_FUELLER_LIFEBIT SpI 009 KEG Füller Lebensbit
      CALL FC    14 (
           UnitNo                   := #UnitNo,
           SpIRec                   := DB2631.KEG_FUELLER_LIFEBIT,
           SpIBit                   := I    986.0);

// KEG_MIXER_LIFEBIT SpI 010 KEG Mixer Lebensbit
      CALL FC    14 (
           UnitNo                   := #UnitNo,
           SpIRec                   := DB2631.KEG_MIXER_LIFEBIT,
           SpIBit                   := I    946.0);

// KEG_MIXER_FRG_CIP_PUMPE SpI 013 KEG Mixer/KZE Freigabe CIP Pumpe
      CALL FC    14 (
           UnitNo                   := #UnitNo,
           SpIRec                   := DB2631.KEG_MIXER_FRG_CIP_PUMPE,
           SpIBit                   := I    946.4);

// KEG_MIXER_FRG_UEBERBR SpI 018 KEG Mixer/KZE Freigabe Überbrückt (Schlüsselschalter)
      CALL FC    14 (
           UnitNo                   := #UnitNo,
           SpIRec                   := DB2631.KEG_MIXER_FRG_UEBERBR,
           SpIBit                   := I    948.1);

// KEG_MIXER_ZEITHALT SpI 019 KEG Mixer/KZE Zeithalt
      CALL FC    14 (
           UnitNo                   := #UnitNo,
           SpIRec                   := DB2631.KEG_MIXER_ZEITHALT,
           SpIBit                   := I    946.5);

NETWORK
TITLE =messages

      NOP   0;
// msg001 Msg 001 Message 01
      CALL FC    16 (
           UnitNo                   := #UnitNo,
           MsgRec                   := DB2637.msg001,
           MsgBit                   := DB2637.DBX   82.7);

// msg002 Msg 002 Message 02
      CALL FC    16 (
           UnitNo                   := #UnitNo,
           MsgRec                   := DB2637.msg002,
           MsgBit                   := DB2637.DBX  142.7);

// msg003 Msg 003 Message 03
      CALL FC    16 (
           UnitNo                   := #UnitNo,
           MsgRec                   := DB2637.msg003,
           MsgBit                   := DB2637.DBX  202.7);

NETWORK
TITLE =unit supply

      UC    FB [#UnitFB];
NETWORK
TITLE =KEG_MIXER_FREIGABE_EIN  KEG Mixer/KZE Freigabe ist eingeschaltet
// Act 001
// Box           : KEG Mixer
// Output address: Q948.1
      CALL FC    70 (
           UnitNo                   := #UnitNo,
           ActRec                   := DB2630.KEG_MIXER_FREIGABE_EIN,
           Typ                      := 0,
           FBa                      := #xTmp,
           FBa2                     := #xTmp,
           Out                      := Q    948.1);

NETWORK
TITLE =KEG_FUELLER_UML_FW  KEG Füller CIP Umlauf Frischwasser
// Act 004
// Box           : KEG Füller
// Output address: Q987.0
      CALL FC    70 (
           UnitNo                   := #UnitNo,
           ActRec                   := DB2630.KEG_FUELLER_UML_FW,
           Typ                      := 0,
           FBa                      := #xTmp,
           FBa2                     := #xTmp,
           Out                      := Q    987.0);

NETWORK
TITLE =KEG_FUELLER_UML_HW  KEG Füller CIP Umlauf HW
// Act 005
// Box           : KEG Füller
// Output address: Q987.1
      CALL FC    70 (
           UnitNo                   := #UnitNo,
           ActRec                   := DB2630.KEG_FUELLER_UML_HW,
           Typ                      := 0,
           FBa                      := #xTmp,
           FBa2                     := #xTmp,
           Out                      := Q    987.1);

NETWORK
TITLE =KEG_FUELLER_UML_LAUGE  KEG Füller CIP Umlauf Lauge
// Act 006
// Box           : KEG Füller
// Output address: Q987.2
      CALL FC    70 (
           UnitNo                   := #UnitNo,
           ActRec                   := DB2630.KEG_FUELLER_UML_LAUGE,
           Typ                      := 0,
           FBa                      := #xTmp,
           FBa2                     := #xTmp,
           Out                      := Q    987.2);

NETWORK
TITLE =KEG_FUELLER_UML_SAEURE  KEG Füller CIP Umlauf Säure
// Act 007
// Box           : KEG Füller
// Output address: Q987.3
      CALL FC    70 (
           UnitNo                   := #UnitNo,
           ActRec                   := DB2630.KEG_FUELLER_UML_SAEURE,
           Typ                      := 0,
           FBa                      := #xTmp,
           FBa2                     := #xTmp,
           Out                      := Q    987.3);

NETWORK
TITLE =KEG_FUELLER_UML_RW  KEG Füller CIP Umlauf Reinwasser
// Act 008
// Box           : KEG Füller
// Output address: Q987.4
      CALL FC    70 (
           UnitNo                   := #UnitNo,
           ActRec                   := DB2630.KEG_FUELLER_UML_RW,
           Typ                      := 0,
           FBa                      := #xTmp,
           FBa2                     := #xTmp,
           Out                      := Q    987.4);

NETWORK
TITLE =KEG_FUELLER_BUS_UEBERW  KEG Füller Bus Überwachung
// Act 009
// Box           : KEG Füller
// Output address: Q987.7
      CALL FC    70 (
           UnitNo                   := #UnitNo,
           ActRec                   := DB2630.KEG_FUELLER_BUS_UEBERW,
           Typ                      := 0,
           FBa                      := #xTmp,
           FBa2                     := #xTmp,
           Out                      := Q    987.7);

NETWORK
TITLE =KEG_FUELLER_BEFUELL  KEG Füller Füllmaschine mit CIP Medium befülle
// Act 010
// Box           : KEG Füller
// Output address: Q986.2
      CALL FC    70 (
           UnitNo                   := #UnitNo,
           ActRec                   := DB2630.KEG_FUELLER_BEFUELL,
           Typ                      := 0,
           FBa                      := #xTmp,
           FBa2                     := #xTmp,
           Out                      := Q    986.2);

NETWORK
TITLE =KEG_MIXER_UML_FW  KEG Mixer/KZE CIP Umlauf Frischwasser
// Act 013
// Box           : KEG Mixer
// Output address: Q947.0
      CALL FC    70 (
           UnitNo                   := #UnitNo,
           ActRec                   := DB2630.KEG_MIXER_UML_FW,
           Typ                      := 0,
           FBa                      := #xTmp,
           FBa2                     := #xTmp,
           Out                      := Q    947.0);

NETWORK
TITLE =KEG_FUELLER_AUSSCH  KEG Füller Füllmaschine mit Luft ausschieben/en
// Act 014
// Box           : KEG Füller
// Output address: Q986.3
      CALL FC    70 (
           UnitNo                   := #UnitNo,
           ActRec                   := DB2630.KEG_FUELLER_AUSSCH,
           Typ                      := 0,
           FBa                      := #xTmp,
           FBa2                     := #xTmp,
           Out                      := Q    986.3);

NETWORK
TITLE =KEG_MIXER_UML_RW  KEG Mixer/KZE CIP Umlauf Reinwasser
// Act 017
// Box           : KEG Mixer
// Output address: Q947.4
      CALL FC    70 (
           UnitNo                   := #UnitNo,
           ActRec                   := DB2630.KEG_MIXER_UML_RW,
           Typ                      := 0,
           FBa                      := #xTmp,
           FBa2                     := #xTmp,
           Out                      := Q    947.4);

NETWORK
TITLE =KEG_MIXER_CIP_LAUGE  KEG Mixer/KZE CIP Programm mit Lauge angewählt
// Act 020
// Box           : KEG Mixer
// Output address: Q946.7
      CALL FC    70 (
           UnitNo                   := #UnitNo,
           ActRec                   := DB2630.KEG_MIXER_CIP_LAUGE,
           Typ                      := 0,
           FBa                      := #xTmp,
           FBa2                     := #xTmp,
           Out                      := Q    946.7);

NETWORK
TITLE =KEG_RR2  CIP Rücklaufventil Kreis 2 KEG Anlage
// Act 021
// Box           : VS-RRA
// Input address : I201.4
// Output address: Q201.4
      CALL FC    70 (
           UnitNo                   := #UnitNo,
           ActRec                   := DB2630.KEG_RR2,
           Typ                      := 1,
           FBa                      := #xTmp,
           FBa2                     := I    201.4,
           Out                      := Q    201.4);

NETWORK
TITLE =KEG_MIXER_UML_LAUGE  KEG Mixer/KZE CIP Umlauf Lauge
// Act 024
// Box           : KEG Mixer
// Output address: Q947.2
      CALL FC    70 (
           UnitNo                   := #UnitNo,
           ActRec                   := DB2630.KEG_MIXER_UML_LAUGE,
           Typ                      := 0,
           FBa                      := #xTmp,
           FBa2                     := #xTmp,
           Out                      := Q    947.2);

NETWORK
TITLE =KEG_MIXER_UML_SAEURE  KEG Mixer/KZE CIP Umlauf Säure
// Act 025
// Box           : KEG Mixer
// Output address: Q947.3
      CALL FC    70 (
           UnitNo                   := #UnitNo,
           ActRec                   := DB2630.KEG_MIXER_UML_SAEURE,
           Typ                      := 0,
           FBa                      := #xTmp,
           FBa2                     := #xTmp,
           Out                      := Q    947.3);

NETWORK
TITLE =KEG_MIXER_UML_HW  KEG Mixer/KZE CIP Umlauf HW
// Act 026
// Box           : KEG Mixer
// Output address: Q947.1
      CALL FC    70 (
           UnitNo                   := #UnitNo,
           ActRec                   := DB2630.KEG_MIXER_UML_HW,
           Typ                      := 0,
           FBa                      := #xTmp,
           FBa2                     := #xTmp,
           Out                      := Q    947.1);

NETWORK
TITLE =KEG_MIXER_FLUTEN  KEG Mixer/KZE Mixer fluten für Standdesinfektion
// Act 027
// Box           : KEG Mixer
// Output address: Q946.2
      CALL FC    70 (
           UnitNo                   := #UnitNo,
           ActRec                   := DB2630.KEG_MIXER_FLUTEN,
           Typ                      := 0,
           FBa                      := #xTmp,
           FBa2                     := #xTmp,
           Out                      := Q    946.2);

NETWORK
TITLE =KEG_MIXER_AUSPUMPEN  KEG Mixer/KZE PDL auspumpen
// Act 030
// Box           : KEG Mixer
// Output address: Q946.3
      CALL FC    70 (
           UnitNo                   := #UnitNo,
           ActRec                   := DB2630.KEG_MIXER_AUSPUMPEN,
           Typ                      := 0,
           FBa                      := #xTmp,
           FBa2                     := #xTmp,
           Out                      := Q    946.3);

NETWORK
TITLE =KEG_FUELLER_CIP_ENDE  KEG Füller CIP Ende
// Act 032
// Box           : KEG Füller
// Output address: Q986.1
      CALL FC    70 (
           UnitNo                   := #UnitNo,
           ActRec                   := DB2630.KEG_FUELLER_CIP_ENDE,
           Typ                      := 0,
           FBa                      := #xTmp,
           FBa2                     := #xTmp,
           Out                      := Q    986.1);

NETWORK
TITLE =KEG_MIXER_CIP_ENDE  KEG Mixer/KZE CIP Ende
// Act 033
// Box           : KEG Mixer
// Output address: Q946.1
      CALL FC    70 (
           UnitNo                   := #UnitNo,
           ActRec                   := DB2630.KEG_MIXER_CIP_ENDE,
           Typ                      := 0,
           FBa                      := #xTmp,
           FBa2                     := #xTmp,
           Out                      := Q    946.1);

NETWORK
TITLE =KEG_MIXER_CIP_PPE_LAEUFT  KEG Mixer/KZE CIP Pumpe läuft
// Act 034
// Box           : KEG Mixer
// Output address: Q946.4
      CALL FC    70 (
           UnitNo                   := #UnitNo,
           ActRec                   := DB2630.KEG_MIXER_CIP_PPE_LAEUFT,
           Typ                      := 0,
           FBa                      := #xTmp,
           FBa2                     := #xTmp,
           Out                      := Q    946.4);

NETWORK
TITLE =Act036  Spare
// Act 036
// Box           : KEG Mixer
// Output address: #DummyBool
      CALL FC    70 (
           UnitNo                   := #UnitNo,
           ActRec                   := DB2630.Act036,
           Typ                      := 0,
           FBa                      := #xTmp,
           FBa2                     := #xTmp,
           Out                      := #DummyBool);

END_FUNCTION_BLOCK

FUNCTION_BLOCK FB 1631
TITLE =U063: Abfüllanlage  3
FAMILY : BOTEC_F1
NAME : U063E
VERSION : 1.2


VAR_TEMP
  CIP : BOOL ;	//CIP active
  UNIM : BOOL ;	//Unit Not In Maintenance
  GenRel : BOOL ;	//general OK (emergency and maintenance OK)
  EStopOK : BOOL ;	//emergency OK
  UnitNo : INT ;	//unit number
  xTmp : BOOL ;	//Temporary Bool
  iTmp : INT ;	//Temporary INT
  rTmp : REAL ;	//Temporary REAL
  dTmp : DINT ;	//Temporary DINT (free for general use)
  RetValInt : INT ;	//return value
END_VAR
BEGIN
NETWORK
TITLE =General

      SET   ;
// Simulation ---------------------------------------------------------------
      A     DB1631.DBX 1357.7;
      CC    FB  1639; // "U063Sim"
      A     DB1631.DBX   17.3;
      =     DB1631.DBX 1357.7; //Help bit for simulation

// get unit number ----------------------------------------------------------
      L     DB1630.DBW    0;
      T     #UnitNo;

// CIP ----------------------------------------------------------------------
      L     DB1631.DBD   54;
      L     0;
      <D    ;
      =     #CIP;

// emergency OK -------------------------------------------------------------
      A     DB1635.DBX   27.0; //Emergency Stop OK
      =     #EStopOK;

// Write Unit in Maintenance ------------------------------------------------

      AN    DB1631.DBX   69.7;
      =     #UNIM;

// emergency and maintenance OK ---------------------------------------------
      A     #EStopOK;
      A     #UNIM;
      =     #GenRel;

// communication ------------------------------------------------------------
      UC    FB  1635; // U063Com

NETWORK
TITLE =Analog Inputs

      NOP   0;

// ----------------------------------------------------------
// KEG_MIXER_KZE_NIVEAU KEG Mixer/KZE Niveau Steriltank
// ----------------------------------------------------------
      L     DB1631.DBD 1118; // !!! insert correct SFM !!!
      T     DB2633.DBD  238;

      SET   ;
      =     DB2633.DBX  141.5;

// ----------------------------------------------------------
// KEG_MIXER_KZE_SORTE KEG Mixer/KZE Sortennummer Produkt
// ----------------------------------------------------------
      L     DB1631.DBD 1118; // !!! insert correct SFM !!!
      T     DB2633.DBD  358;

      SET   ;
      =     DB2633.DBX  261.5;

NETWORK
TITLE =Universal Value

      NOP   0;

// ----------------------------------------------------------
// unv001 Process Status
// ----------------------------------------------------------
// process value to UnV
//      L     0.000000e+000
//      T     "U063UnVD".unv001.ValExt

// ----------------------------------------------------------
// unv002 Universal Value 02
// ----------------------------------------------------------
// process value to UnV
//      L     0.000000e+000
//      T     "U063UnVD".unv002.ValExt

// ----------------------------------------------------------
// KEG_MIXER_PROGRAMMNR Preselection 1/2/3 GES./GES.without KZE/KZE
// ----------------------------------------------------------
// process value to UnV
//      L     0.000000e+000
//      T     "U063UnVD".KEG_MIXER_PROGRAMMNR.ValExt

// ----------------------------------------------------------
// KEG_MIXER_TANKNUMMER Tank number clean water tank [1..9]
// ----------------------------------------------------------
// process value to UnV
//      L     0.000000e+000
//      T     "U063UnVD".KEG_MIXER_TANKNUMMER.ValExt

NETWORK
TITLE =Special Input

      NOP   0;

// ----------------------------------------------------------
// KEG_MIXER_CIP_BEREIT KEG Mixer/KZE CIP Bereit
// ----------------------------------------------------------
//      CLR
//      =     "U063SpID".KEG_MIXER_CIP_BEREIT.EAl
//      =     "U063SpID".KEG_MIXER_CIP_BEREIT.Pre

// ----------------------------------------------------------
// KEG_MIXER_VOLL KEG Mixer/KZE Vollmeldung
// ----------------------------------------------------------
//      CLR
//      =     "U063SpID".KEG_MIXER_VOLL.EAl
//      =     "U063SpID".KEG_MIXER_VOLL.Pre

// ----------------------------------------------------------
// KEG_MIXER_LEER KEG Mixer/KZE Leermeldung
// ----------------------------------------------------------
//      CLR
//      =     "U063SpID".KEG_MIXER_LEER.EAl
//      =     "U063SpID".KEG_MIXER_LEER.Pre

// ----------------------------------------------------------
// KEG_FUELLER_CIP_BEREIT KEG Füller CIP Bereitschaft
// ----------------------------------------------------------
//      CLR
//      =     "U063SpID".KEG_FUELLER_CIP_BEREIT.EAl
//      =     "U063SpID".KEG_FUELLER_CIP_BEREIT.Pre

// ----------------------------------------------------------
// KEG_FUELLER_LIFEBIT KEG Füller Lebensbit
// ----------------------------------------------------------
//      CLR
//      =     "U063SpID".KEG_FUELLER_LIFEBIT.EAl
//      =     "U063SpID".KEG_FUELLER_LIFEBIT.Pre

// ----------------------------------------------------------
// KEG_MIXER_LIFEBIT KEG Mixer Lebensbit
// ----------------------------------------------------------
//      CLR
//      =     "U063SpID".KEG_MIXER_LIFEBIT.EAl
//      =     "U063SpID".KEG_MIXER_LIFEBIT.Pre

// ----------------------------------------------------------
// KEG_MIXER_FRG_CIP_PUMPE KEG Mixer/KZE Freigabe CIP Pumpe
// ----------------------------------------------------------
//      CLR
//      =     "U063SpID".KEG_MIXER_FRG_CIP_PUMPE.EAl
//      =     "U063SpID".KEG_MIXER_FRG_CIP_PUMPE.Pre

// ----------------------------------------------------------
// KEG_MIXER_FRG_UEBERBR KEG Mixer/KZE Freigabe Überbrückt (Schlüsselschalter)
// ----------------------------------------------------------
//      CLR
//      =     "U063SpID".KEG_MIXER_FRG_UEBERBR.EAl
//      =     "U063SpID".KEG_MIXER_FRG_UEBERBR.Pre

// ----------------------------------------------------------
// KEG_MIXER_ZEITHALT KEG Mixer/KZE Zeithalt
// ----------------------------------------------------------
//      CLR
//      =     "U063SpID".KEG_MIXER_ZEITHALT.EAl
//      =     "U063SpID".KEG_MIXER_ZEITHALT.Pre

NETWORK
TITLE =Messages

      NOP   0;

// ----------------------------------------------------------
// msg001 Message 01
// ----------------------------------------------------------
      SET   ;
      R     DB2637.DBX   80.7;
      =     DB2637.DBX   81.4;

      CLR   ;
      =     DB2637.DBX   82.7;

// ----------------------------------------------------------
// msg002 Message 02
// ----------------------------------------------------------
      SET   ;
      R     DB2637.DBX  140.7;
      =     DB2637.DBX  141.4;

      CLR   ;
      =     DB2637.DBX  142.7;

// ----------------------------------------------------------
// msg003 Message 03
// ----------------------------------------------------------
      SET   ;
      R     DB2637.DBX  200.7;
      =     DB2637.DBX  201.4;

      CLR   ;
      =     DB2637.DBX  202.7;

NETWORK
TITLE =Sequence organisation

      CLR   ;
      =     M    122.2;

// SFM supply ----------------------------------------------------------------

// analog value to SFM KEG Mixer/KZE Niveau Steriltank  -----------------------
      L     DB2633.DBD  146;
      T     DB1631.DBD 1122; // !!! insert correct SFM !!!

// analog value to SFM KEG Mixer/KZE Sortennummer Produkt -----------------------
      L     DB2633.DBD  266;
      T     DB1631.DBD 1122; // !!! insert correct SFM !!!

// sequencer ----------------------------------------------------------------
      A     DB1633.DBX   43.1;
      S     DB1633.DBX   97.3;

      CALL FC    40 (
           UnitNo                   := #UnitNo);

NETWORK
TITLE =Auto / Manual

      SET   ;
      AN    M    122.2;
      JC    MODE;
      AN    M    120.1;

// assign actuator mode
      AN    M    120.1;
      =     DB2630.DBX  105.4;
      =     DB2630.DBX  345.4;
      =     DB2630.DBX  425.4;
      =     DB2630.DBX  505.4;
      =     DB2630.DBX  585.4;
      =     DB2630.DBX  665.4;
      =     DB2630.DBX  745.4;
      =     DB2630.DBX  825.4;
      =     DB2630.DBX 1065.4;
      =     DB2630.DBX 1145.4;
      =     DB2630.DBX 1385.4;
      =     DB2630.DBX 1625.4;
      =     DB2630.DBX 1705.4;
      =     DB2630.DBX 1945.4;
      =     DB2630.DBX 2025.4;
      =     DB2630.DBX 2105.4;
      =     DB2630.DBX 2185.4;
      =     DB2630.DBX 2425.4;
      =     DB2630.DBX 2585.4;
      =     DB2630.DBX 2665.4;
      =     DB2630.DBX 2745.4;
      =     DB2630.DBX 2905.4;



MODE: SET   ;

NETWORK
TITLE =KEG_MIXER_FREIGABE_EIN KEG Mixer/KZE Freigabe ist eingeschaltet
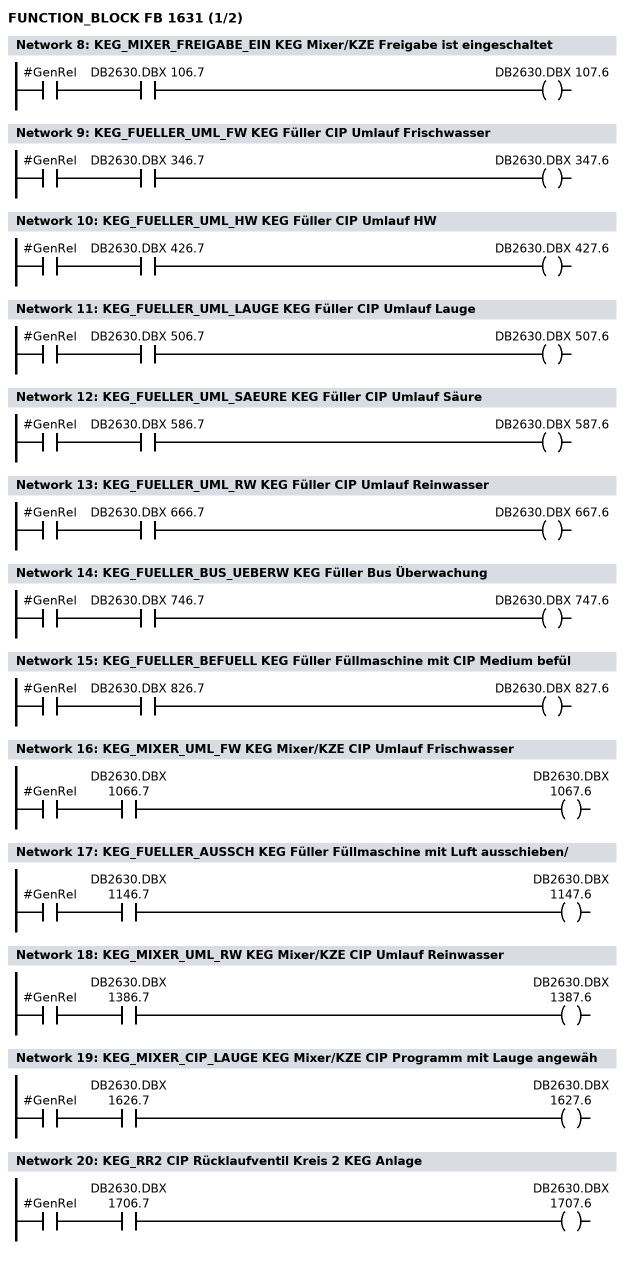

      A     #GenRel;
      A     DB2630.DBX  106.7;
      =     DB2630.DBX  107.6;
NETWORK
TITLE =KEG_FUELLER_UML_FW KEG Füller CIP Umlauf Frischwasser

      A     #GenRel;
      A     DB2630.DBX  346.7;
      =     DB2630.DBX  347.6;
NETWORK
TITLE =KEG_FUELLER_UML_HW KEG Füller CIP Umlauf HW

      A     #GenRel;
      A     DB2630.DBX  426.7;
      =     DB2630.DBX  427.6;
NETWORK
TITLE =KEG_FUELLER_UML_LAUGE KEG Füller CIP Umlauf Lauge

      A     #GenRel;
      A     DB2630.DBX  506.7;
      =     DB2630.DBX  507.6;
NETWORK
TITLE =KEG_FUELLER_UML_SAEURE KEG Füller CIP Umlauf Säure

      A     #GenRel;
      A     DB2630.DBX  586.7;
      =     DB2630.DBX  587.6;
NETWORK
TITLE =KEG_FUELLER_UML_RW KEG Füller CIP Umlauf Reinwasser

      A     #GenRel;
      A     DB2630.DBX  666.7;
      =     DB2630.DBX  667.6;
NETWORK
TITLE =KEG_FUELLER_BUS_UEBERW KEG Füller Bus Überwachung

      A     #GenRel;
      A     DB2630.DBX  746.7;
      =     DB2630.DBX  747.6;
NETWORK
TITLE =KEG_FUELLER_BEFUELL KEG Füller Füllmaschine mit CIP Medium befül

      A     #GenRel;
      A     DB2630.DBX  826.7;
      =     DB2630.DBX  827.6;
NETWORK
TITLE =KEG_MIXER_UML_FW KEG Mixer/KZE CIP Umlauf Frischwasser

      A     #GenRel;
      A     DB2630.DBX 1066.7;
      =     DB2630.DBX 1067.6;
NETWORK
TITLE =KEG_FUELLER_AUSSCH KEG Füller Füllmaschine mit Luft ausschieben/

      A     #GenRel;
      A     DB2630.DBX 1146.7;
      =     DB2630.DBX 1147.6;
NETWORK
TITLE =KEG_MIXER_UML_RW KEG Mixer/KZE CIP Umlauf Reinwasser

      A     #GenRel;
      A     DB2630.DBX 1386.7;
      =     DB2630.DBX 1387.6;
NETWORK
TITLE =KEG_MIXER_CIP_LAUGE KEG Mixer/KZE CIP Programm mit Lauge angewäh

      A     #GenRel;
      A     DB2630.DBX 1626.7;
      =     DB2630.DBX 1627.6;
NETWORK
TITLE =KEG_RR2 CIP Rücklaufventil Kreis 2 KEG Anlage

      A     #GenRel;
      A     DB2630.DBX 1706.7;
      =     DB2630.DBX 1707.6;
NETWORK
TITLE =KEG_MIXER_UML_LAUGE KEG Mixer/KZE CIP Umlauf Lauge
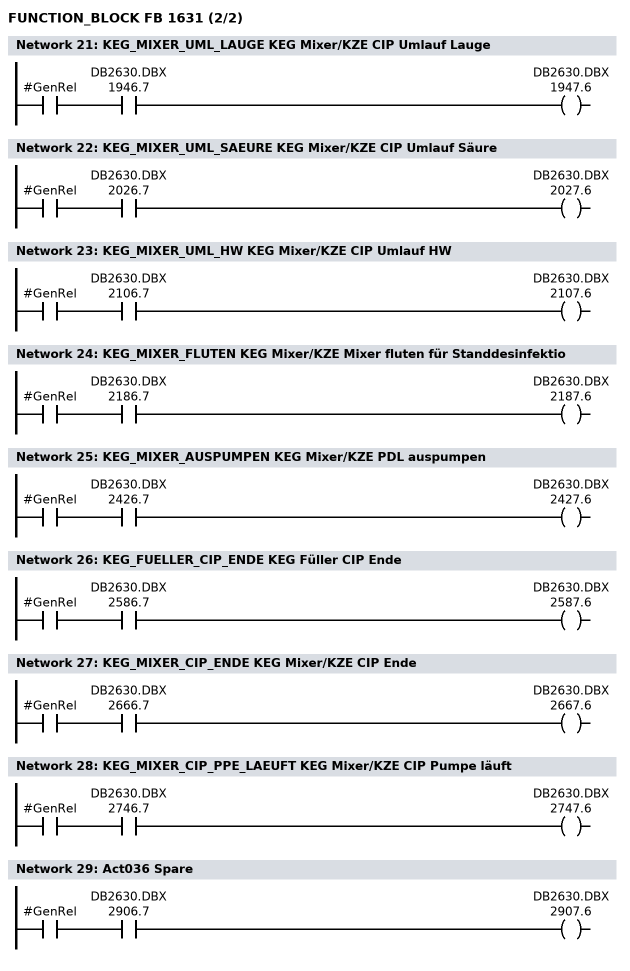

      A     #GenRel;
      A     DB2630.DBX 1946.7;
      =     DB2630.DBX 1947.6;
NETWORK
TITLE =KEG_MIXER_UML_SAEURE KEG Mixer/KZE CIP Umlauf Säure

      A     #GenRel;
      A     DB2630.DBX 2026.7;
      =     DB2630.DBX 2027.6;
NETWORK
TITLE =KEG_MIXER_UML_HW KEG Mixer/KZE CIP Umlauf HW

      A     #GenRel;
      A     DB2630.DBX 2106.7;
      =     DB2630.DBX 2107.6;
NETWORK
TITLE =KEG_MIXER_FLUTEN KEG Mixer/KZE Mixer fluten für Standdesinfektio

      A     #GenRel;
      A     DB2630.DBX 2186.7;
      =     DB2630.DBX 2187.6;
NETWORK
TITLE =KEG_MIXER_AUSPUMPEN KEG Mixer/KZE PDL auspumpen

      A     #GenRel;
      A     DB2630.DBX 2426.7;
      =     DB2630.DBX 2427.6;
NETWORK
TITLE =KEG_FUELLER_CIP_ENDE KEG Füller CIP Ende

      A     #GenRel;
      A     DB2630.DBX 2586.7;
      =     DB2630.DBX 2587.6;
NETWORK
TITLE =KEG_MIXER_CIP_ENDE KEG Mixer/KZE CIP Ende

      A     #GenRel;
      A     DB2630.DBX 2666.7;
      =     DB2630.DBX 2667.6;
NETWORK
TITLE =KEG_MIXER_CIP_PPE_LAEUFT KEG Mixer/KZE CIP Pumpe läuft

      A     #GenRel;
      A     DB2630.DBX 2746.7;
      =     DB2630.DBX 2747.6;
NETWORK
TITLE =Act036 Spare

      A     #GenRel;
      A     DB2630.DBX 2906.7;
      =     DB2630.DBX 2907.6;
END_FUNCTION_BLOCK

FUNCTION_BLOCK FB 1650
TITLE =U065: Abfüllanlage  5
FAMILY : BOTEC_F1
NAME : U065A
VERSION : 2.1


VAR_TEMP
  EStopOK : BOOL ;	//auxiliary flag
  CIP : BOOL ;	//CIP Program Selected
  xTmp : BOOL ;	//Temporary Bool(free for general use)
  DummyBool : BOOL ;	//Temporary Bool(free for general use)
  UnitNo : INT ;	//unit number
  UnitFB : INT ;	//unit expansion FB number
  rTmp : REAL ;	//Temporary REAL (free for general use)
  iTmp : INT ;	//Temporary INT (free for general use)
  DummyInt : INT ;	//Temporary INT (free for general use)
  dTmp : DINT ;	//Temporary DINT (free for general use)
END_VAR
BEGIN
NETWORK
TITLE =general

      CLR   ;
      =     #xTmp;
      =     #EStopOK;

      L     DB1650.DBW    0;
      T     #UnitNo;
      L     DB1650.DBW    2;
      T     #UnitFB;

NETWORK
TITLE =analog inputs

      NOP   0;
// A5_TI1 AnI 001
      CALL FC    24 (
           UnitNo                   := #UnitNo,
           AnIRec                   := DB2653.A5_TI1,
           ValPer                   := PIW  512);

NETWORK
TITLE =Universal value

      NOP   0;
// unv001 UnV 001 Process Status
      CALL FC    27 (
           UnitNo                   := #UnitNo,
           UnVRec                   := DB2655.unv001,
           ValExt                   := DB2655.DBD  234);

// unv002 UnV 002 Universal Value 02
      CALL FC    27 (
           UnitNo                   := #UnitNo,
           UnVRec                   := DB2655.unv002,
           ValExt                   := DB2655.DBD  362);

// unv003 UnV 003 Universal Value 03
      CALL FC    27 (
           UnitNo                   := #UnitNo,
           UnVRec                   := DB2655.unv003,
           ValExt                   := DB2655.DBD  490);

// unv004 UnV 004 Universal Value 04
      CALL FC    27 (
           UnitNo                   := #UnitNo,
           UnVRec                   := DB2655.unv004,
           ValExt                   := DB2655.DBD  618);

NETWORK
TITLE =special inputs

      NOP   0;
// A5_FS1 SpI 001 Anlage 5 Strömungswächter
      CALL FC    14 (
           UnitNo                   := #UnitNo,
           SpIRec                   := DB2651.A5_FS1,
           SpIBit                   := I    195.0);

// A5_FUELLER_LAEUFT SpI 002 Koppelsignal von Füller 5 Füller läuft (Dauersignal)
      CALL FC    14 (
           UnitNo                   := #UnitNo,
           SpIRec                   := DB2651.A5_FUELLER_LAEUFT,
           SpIBit                   := I    196.1);

// A5_MIXER_CIP_BEREIT SpI 003 Koppelsignal von Mixer 5 CIP-Bereitschaft (Dauersignal)
      CALL FC    14 (
           UnitNo                   := #UnitNo,
           SpIRec                   := DB2651.A5_MIXER_CIP_BEREIT,
           SpIBit                   := I    198.0);

// A5_MIXER_VOLL SpI 004 Koppelsignal von Mixer 5 Mixer voll
      CALL FC    14 (
           UnitNo                   := #UnitNo,
           SpIRec                   := DB2651.A5_MIXER_VOLL,
           SpIBit                   := I    198.1);

// A5_MIXER_LEER SpI 005 Koppelsignal von Mixer 5 Mixer leer
      CALL FC    14 (
           UnitNo                   := #UnitNo,
           SpIRec                   := DB2651.A5_MIXER_LEER,
           SpIBit                   := I    198.2);

// A5_MIXER_Anforderung SpI 006 Koppelsignal von Mixer 5 Anforderung Nachsp.
      CALL FC    14 (
           UnitNo                   := #UnitNo,
           SpIRec                   := DB2651.A5_MIXER_Anforderung,
           SpIBit                   := I    198.3);

// A5_FUELLER_CIP_BEREIT SpI 007 Koppelsignal von Füller 5 CIP-Bereitschaft (Dauersignal)
      CALL FC    14 (
           UnitNo                   := #UnitNo,
           SpIRec                   := DB2651.A5_FUELLER_CIP_BEREIT,
           SpIBit                   := I    196.0);

// F5_WATCHDOG SpI 009 Koppelsignal von Füller 5 WATCHDOG
      CALL FC    14 (
           UnitNo                   := #UnitNo,
           SpIRec                   := DB2651.F5_WATCHDOG,
           SpIBit                   := I    197.7);

// M5_WATCHDOG SpI 010 Koppelsignal von Mixer 5 WATCHDOG
      CALL FC    14 (
           UnitNo                   := #UnitNo,
           SpIRec                   := DB2651.M5_WATCHDOG,
           SpIBit                   := I    199.7);

// A5_FUELLER_LEER SpI 011 Koppelsignal von Füller 5 Füller leer (Impuls)
      CALL FC    14 (
           UnitNo                   := #UnitNo,
           SpIRec                   := DB2651.A5_FUELLER_LEER,
           SpIBit                   := I    196.2);

// A5_FUELLER_VOLL SpI 012 Koppelsignal von Füller 5 Füller voll (Impuls)
      CALL FC    14 (
           UnitNo                   := #UnitNo,
           SpIRec                   := DB2651.A5_FUELLER_VOLL,
           SpIBit                   := I    196.3);

// A5_RINSER_CIP_BEREIT SpI 013 Koppelsignal von Rinser 5 CIP-Bereitschaft (Dauersignal)
      CALL FC    14 (
           UnitNo                   := #UnitNo,
           SpIRec                   := DB2651.A5_RINSER_CIP_BEREIT,
           SpIBit                   := I    172.0);

// A5_RINSER_LAEUFT SpI 014 Koppelsignal von Rinser 5 Rinser läuft (Dauersignal)
      CALL FC    14 (
           UnitNo                   := #UnitNo,
           SpIRec                   := DB2651.A5_RINSER_LAEUFT,
           SpIBit                   := I    172.1);

// R5_WATCHDOG SpI 015 Koppelsignal von Rinser 5 WATCHDOG
      CALL FC    14 (
           UnitNo                   := #UnitNo,
           SpIRec                   := DB2651.R5_WATCHDOG,
           SpIBit                   := I    173.7);

// GOA503 SpI 017 MOLCH A5 GOA503
      CALL FC    14 (
           UnitNo                   := #UnitNo,
           SpIRec                   := DB2651.GOA503,
           SpIBit                   := I    194.2);

// A5_FUELLER_KLARSPUELEN SpI 018 Koppelsignal von Füller 5 Klarspülen
      CALL FC    14 (
           UnitNo                   := #UnitNo,
           SpIRec                   := DB2651.A5_FUELLER_KLARSPUELEN,
           SpIBit                   := I    196.4);

NETWORK
TITLE =messages

      NOP   0;
// msg001 Msg 001 Message 01
      CALL FC    16 (
           UnitNo                   := #UnitNo,
           MsgRec                   := DB2657.msg001,
           MsgBit                   := DB2657.DBX   82.7);

// msg002 Msg 002 Message 02
      CALL FC    16 (
           UnitNo                   := #UnitNo,
           MsgRec                   := DB2657.msg002,
           MsgBit                   := DB2657.DBX  142.7);

// msg003 Msg 003 Message 03
      CALL FC    16 (
           UnitNo                   := #UnitNo,
           MsgRec                   := DB2657.msg003,
           MsgBit                   := DB2657.DBX  202.7);

NETWORK
TITLE =unit supply

      UC    FB [#UnitFB];

NETWORK
TITLE =A5_RP1  Rücklaufpumpe Anlage 5
// Act 001
// Box           : S6 U6.3
// Input address : I5.2
// Output address: Q5.2
      CALL FC    70 (
           UnitNo                   := #UnitNo,
           ActRec                   := DB2650.A5_RP1,
           Typ                      := 1,
           FBa                      := #xTmp,
           FBa2                     := I      5.2,
           Out                      := Q      5.2);

NETWORK
TITLE =F5_Maschine_Start  Füller A5 Maschine Start
// Act 002
// Box           : Füller5
// Output address: Q196.0
      CALL FC    70 (
           UnitNo                   := #UnitNo,
           ActRec                   := DB2650.F5_Maschine_Start,
           Typ                      := 0,
           FBa                      := #xTmp,
           FBa2                     := #xTmp,
           Out                      := Q    196.0);

NETWORK
TITLE =F5_Maschine_Stop  Füller A5 Maschine Stop
// Act 003
// Box           : Füller5
// Output address: Q196.1
      CALL FC    70 (
           UnitNo                   := #UnitNo,
           ActRec                   := DB2650.F5_Maschine_Stop,
           Typ                      := 0,
           FBa                      := #xTmp,
           FBa2                     := #xTmp,
           Out                      := #xTmp);

NETWORK
TITLE =R5_START  Rinser A5 Maschine Start
// Act 004
// Box           : Rinser5
// Output address: Q172.0
      CALL FC    70 (
           UnitNo                   := #UnitNo,
           ActRec                   := DB2650.R5_START,
           Typ                      := 0,
           FBa                      := #xTmp,
           FBa2                     := #xTmp,
           Out                      := Q    172.0);

NETWORK
TITLE =R5_STOP  Rinser A5 Maschine Stop
// Act 005
// Box           : Rinser5
// Output address: Q172.1
      CALL FC    70 (
           UnitNo                   := #UnitNo,
           ActRec                   := DB2650.R5_STOP,
           Typ                      := 0,
           FBa                      := #xTmp,
           FBa2                     := #xTmp,
           Out                      := #xTmp);

